# B&R Automation Studio project NAINV104C00R8L515F00 (part 12)

#### Act_OptP0923FullMask.st
```iecst
ACTION Act_OptP0923FullMask:

	IF eCurrPage = UIP0923Stopper THEN

		IF p_tyDI.bEStopSig = FALSE THEN
			p_tyC0002FullMask ACCESS ADR(tyP0923Stopper.tyFullMaskEStop);

		ELSIF p_tyDI.bCoverSWSig = FALSE THEN
			p_tyC0002FullMask ACCESS ADR(tyP0923Stopper.tyFullMaskCWSig);

		ELSIF p_tyDI.bSafetyRlySig = FALSE THEN
			p_tyC0002FullMask ACCESS ADR(tyP0923Stopper.tyFullMaskSafetyRly);

		ELSE
			p_tyC0002FullMask ACCESS ADR(tyP0923Stopper.tyFullMaskHide);

		END_IF

	END_IF

END_ACTION
```

#### Act_OptP0923Navi.st
```iecst
ACTION Act_OptP0923Navi:

	IF tyP0923Stopper.tyNaviBack.tyBtnBack.bRtCompl = TRUE THEN
		tyP0923Stopper.tyNaviBack.tyBtnBack.bRtCompl 	:= FALSE;
		tyP0923Stopper.tyNaviBack.tyBtnBack.bValue		:= FALSE;

		eChgPage	:= UIP0920MtrNPneuCtrl;

	END_IF

END_ACTION
```

#### Act_OptP0923ChgLyr.st
```iecst
ACTION Act_OptP0923ChgLyr:

	IF tyP0923Stopper.tyCom.tyBtnDCCtrl.bRtCompl = TRUE THEN
		tyP0923Stopper.tyCom.tyBtnDCCtrl.bRtCompl := FALSE;

		IF tyP0923Stopper.tyCom.tyBtnDCCtrl.bValue = TRUE THEN
			fUIInRtStatOff(ADR(tyP0923Stopper.tyDC.tyLyr.uiRtStat));
			fUIInRtStatHide(ADR(tyP0923Stopper.tyFB.tyLyr.uiRtStat));
		ELSE
			fUIInRtStatHide(ADR(tyP0923Stopper.tyDC.tyLyr.uiRtStat));
			fUIInRtStatOff(ADR(tyP0923Stopper.tyFB.tyLyr.uiRtStat));
		END_IF
	END_IF

END_ACTION
```

#### Act_OptP0923UpdtData.st
```iecst
ACTION Act_OptP0923UpdtData:

	//Update Bitmap
	IF p_bStopperExtCtrl THEN
		tyP0923Stopper.tyCom.tyBitmapMc.usiValueIdx	:= 1;
	ELSE
		tyP0923Stopper.tyCom.tyBitmapMc.usiValueIdx	:= 0;
	END_IF

END_ACTION
```

#### Act_OptP0923FBCtrl.st
```iecst
ACTION Act_OptP0923FBCtrl:

	IF tyP0923Stopper.tyCom.tyBtnDCCtrl.bValue = FALSE THEN

		//Control
		IF tyP0923Stopper.tyFB.tyBtnRetract.bRtCompl = TRUE THEN
			tyP0923Stopper.tyFB.tyBtnRetract.bRtCompl	:= FALSE;

			tyP0923Stopper.tyFB.tyBtnRetract.bValue		:= TRUE;
			tyP0923Stopper.tyFB.tyBtnExtend.bValue		:= FALSE;

		ELSIF tyP0923Stopper.tyFB.tyBtnExtend.bRtCompl = TRUE THEN
			tyP0923Stopper.tyFB.tyBtnExtend.bRtCompl	:= FALSE;

			tyP0923Stopper.tyFB.tyBtnExtend.bValue		:= TRUE;
			tyP0923Stopper.tyFB.tyBtnRetract.bValue		:= FALSE;

		END_IF

		//Action
		IF tyP0923Stopper.tyFB.tyBtnRetract.bValue = TRUE THEN
			eStopperAct	:= PneuActRet;

			IF p_eStopperStat = PneuActRet AND p_eStopperStatus = Done THEN
				eStopperAct	:= PneuActIdle;

				tyP0923Stopper.tyCom.tyBitmapMc.usiValueIdx	:= 0;
				tyP0923Stopper.tyFB.tyBtnRetract.bValue	:= FALSE;

			ELSIF p_eStopperStatus = Error THEN
				tyP0923Stopper.tyFB.tyBtnRetract.bValue	:= FALSE;

			END_IF

		ELSIF tyP0923Stopper.tyFB.tyBtnExtend.bValue = TRUE THEN
			eStopperAct	:= PneuActExt;

			IF p_eStopperStat = PneuActExt AND p_eStopperStatus = Done THEN
				eStopperAct	:= PneuActIdle;

				tyP0923Stopper.tyCom.tyBitmapMc.usiValueIdx	:= 1;
				tyP0923Stopper.tyFB.tyBtnExtend.bValue := FALSE;

			ELSIF p_eStopperStatus = Error THEN
				tyP0923Stopper.tyFB.tyBtnExtend.bValue := FALSE;

			END_IF
		END_IF

		//Update Status
		tyP0923Stopper.tyDC.tyBtnRetract.bRtCompl	:= FALSE;
		tyP0923Stopper.tyDC.tyBtnExtend.bRtCompl	:= FALSE;
		tyP0923Stopper.tyDC.tyBtnRetract.bValue		:= p_bStopperRetCtrl;
		tyP0923Stopper.tyDC.tyBtnExtend.bValue		:= p_bStopperExtCtrl;

		IF p_tyUsrMgmtCurrAccessRgt.bManualFBOnly THEN
			fUIInRtStatOff(ADR(tyP0923Stopper.tyCom.tyBtnDCCtrl.uiMaskRtStat));
		ELSE
			fUIInRtStatHide(ADR(tyP0923Stopper.tyCom.tyBtnDCCtrl.uiMaskRtStat));
		END_IF

	END_IF

END_ACTION
```

#### Act_OptP0923FBStat.st
```iecst
ACTION Act_OptP0923FBStat:

	tyP0923Stopper.tyFB.tyStringStat.sValue	:= p_sStopperStatTxt;

END_ACTION
```

#### Act_OptP0923DCCtrl.st
```iecst
ACTION Act_OptP0923DCCtrl:

	IF tyP0923Stopper.tyCom.tyBtnDCCtrl.bValue = TRUE THEN

		IF p_bStopperTwoCtrlOut = FALSE THEN

			IF tyP0923Stopper.tyDC.tyBtnRetract.bRtCompl = TRUE THEN
				tyP0923Stopper.tyDC.tyBtnRetract.bValue	:= TRUE;
				tyP0923Stopper.tyDC.tyBtnExtend.bValue	:= FALSE;

				eStopperAct	:= PneuActSetRet;

				IF p_eStopperStat = PneuActSetRet AND p_eStopperStatus = Done THEN
					eStopperAct	:= PneuActIdle;

					tyP0923Stopper.tyCom.tyBitmapMc.usiValueIdx	:= 0;
					tyP0923Stopper.tyDC.tyBtnRetract.bRtCompl	:= FALSE;
				END_IF

			ELSIF tyP0923Stopper.tyDC.tyBtnExtend.bRtCompl = TRUE THEN
				tyP0923Stopper.tyDC.tyBtnExtend.bValue	:= TRUE;
				tyP0923Stopper.tyDC.tyBtnRetract.bValue	:= FALSE;

				eStopperAct	:= PneuActSetExt;

				IF p_eStopperStat = PneuActSetExt AND p_eStopperStatus = Done THEN
					eStopperAct	:= PneuActIdle;

					tyP0923Stopper.tyCom.tyBitmapMc.usiValueIdx	:= 1;
					tyP0923Stopper.tyDC.tyBtnExtend.bRtCompl	:= FALSE;
				END_IF
			END_IF

		ELSE

			IF (tyP0923Stopper.tyDC.tyBtnRetract.bRtCompl = TRUE) OR (tyP0923Stopper.tyDC.tyBtnExtend.bRtCompl = TRUE) THEN
				IF (tyP0923Stopper.tyDC.tyBtnRetract.bValue = TRUE) AND (tyP0923Stopper.tyDC.tyBtnExtend.bValue = TRUE) THEN
					eStopperAct	:= PneuActSetAll;

					IF p_eStopperStat = PneuActSetAll AND p_eStopperStatus = Done THEN
						eStopperAct	:= PneuActIdle;

						tyP0923Stopper.tyDC.tyBtnRetract.bRtCompl	:= FALSE;
						tyP0923Stopper.tyDC.tyBtnExtend.bRtCompl	:= FALSE;
					END_IF

				ELSIF (tyP0923Stopper.tyDC.tyBtnRetract.bValue = TRUE) AND (tyP0923Stopper.tyDC.tyBtnExtend.bValue = FALSE) THEN
					eStopperAct	:= PneuActSetRet;

					IF p_eStopperStat = PneuActSetRet AND p_eStopperStatus = Done THEN
						eStopperAct	:= PneuActIdle;

						tyP0923Stopper.tyCom.tyBitmapMc.usiValueIdx	:= 0;
						tyP0923Stopper.tyDC.tyBtnRetract.bRtCompl	:= FALSE;
						tyP0923Stopper.tyDC.tyBtnExtend.bRtCompl	:= FALSE;
					END_IF

				ELSIF (tyP0923Stopper.tyDC.tyBtnRetract.bValue = FALSE) AND (tyP0923Stopper.tyDC.tyBtnExtend.bValue = TRUE) THEN
					eStopperAct	:= PneuActSetExt;

					IF p_eStopperStat = PneuActSetExt AND p_eStopperStatus = Done THEN
						eStopperAct	:= PneuActIdle;

						tyP0923Stopper.tyCom.tyBitmapMc.usiValueIdx	:= 1;
						tyP0923Stopper.tyDC.tyBtnRetract.bRtCompl	:= FALSE;
						tyP0923Stopper.tyDC.tyBtnExtend.bRtCompl	:= FALSE;
					END_IF

				ELSE
					eStopperAct	:= PneuActRstAll;

					IF p_eStopperStat = PneuActRstAll AND p_eStopperStatus = Done THEN
						eStopperAct	:= PneuActIdle;

						tyP0923Stopper.tyDC.tyBtnRetract.bRtCompl	:= FALSE;
						tyP0923Stopper.tyDC.tyBtnExtend.bRtCompl	:= FALSE;
					END_IF

				END_IF

			END_IF

		END_IF

		tyP0923Stopper.tyFB.tyBtnExtend.bRtCompl	:= FALSE;
		tyP0923Stopper.tyFB.tyBtnExtend.bValue		:= FALSE;
		tyP0923Stopper.tyFB.tyBtnRetract.bRtCompl	:= FALSE;
		tyP0923Stopper.tyFB.tyBtnRetract.bValue		:= FALSE;

	END_IF

END_ACTION
```

#### Act_OptP0923RstMnl.st
```iecst
ACTION Act_OptP0923RstMnl:

	IF EDGEPOS(p_eStopperStatus = Error) THEN

		eStopperAct	:= PneuActIdle;

		tyP0923Stopper.tyDC.tyBtnRetract.bValue 	:= FALSE;
		tyP0923Stopper.tyDC.tyBtnRetract.bRtCompl 	:= FALSE;

		tyP0923Stopper.tyDC.tyBtnExtend.bValue 		:= FALSE;
		tyP0923Stopper.tyDC.tyBtnExtend.bRtCompl 	:= FALSE;

		tyP0923Stopper.tyFB.tyBtnRetract.bValue 	:= FALSE;
		tyP0923Stopper.tyFB.tyBtnRetract.bRtCompl 	:= FALSE;

		tyP0923Stopper.tyFB.tyBtnExtend.bValue 		:= FALSE;
		tyP0923Stopper.tyFB.tyBtnExtend.bRtCompl 	:= FALSE;

	END_IF

	//Reset to Function Block Layer
	IF EDGEPOS(bManualMod = FALSE) THEN
		tyP0923Stopper.tyCom.tyBtnDCCtrl.bValue := FALSE;

		fUIInRtStatHide(ADR(tyP0923Stopper.tyDC.tyLyr.uiRtStat));
		fUIInRtStatOff(ADR(tyP0923Stopper.tyFB.tyLyr.uiRtStat));

		eStopperAct	:= PneuActIdle;

		tyP0923Stopper.tyDC.tyBtnRetract.bValue 	:= FALSE;
		tyP0923Stopper.tyDC.tyBtnRetract.bRtCompl 	:= FALSE;

		tyP0923Stopper.tyDC.tyBtnExtend.bValue 		:= FALSE;
		tyP0923Stopper.tyDC.tyBtnExtend.bRtCompl 	:= FALSE;

		tyP0923Stopper.tyFB.tyBtnRetract.bValue 	:= FALSE;
		tyP0923Stopper.tyFB.tyBtnRetract.bRtCompl 	:= FALSE;

		tyP0923Stopper.tyFB.tyBtnExtend.bValue 		:= FALSE;
		tyP0923Stopper.tyFB.tyBtnExtend.bRtCompl 	:= FALSE;

	END_IF

END_ACTION
```

#### Act_EntP0924Disp.st
```iecst
ACTION Act_EntP0924Disp:

	//Access Address
	p_tyC0003DualMask ACCESS ADR(tyP0924ClampWithRS.tyDualMaskHide);

	p_tyC0004Navi ACCESS ADR(tyP0924ClampWithRS.tyNaviLyr1);

	p_tyC0005Main ACCESS ADR(tyCommon.tyMain);

	p_tyC0007Notif ACCESS ADR(tyCommon.tyNotif);

	p_tyC0008MsgBox ACCESS ADR(tyP0924ClampWithRS.tyMsgBoxHide);

	p_tyC0009Info ACCESS ADR(tyCommon.tyInfo);

	p_tyP0924Clamp1WithRSCom ACCESS ADR(tyP0924ClampWithRS.tyClamp1WithRSCom);
	p_tyP0924Clamp1WithRSDC ACCESS ADR(tyP0924ClampWithRS.tyClamp1WithRSDC);
	p_tyP0924Clamp1WithRSFB ACCESS ADR(tyP0924ClampWithRS.tyClamp1WithRSFB);
	p_tyP0924Clamp1WithRSDis ACCESS ADR(tyP0924ClampWithRS.tyClamp1WithRSDis);

	p_tyP0924Clamp2WithRSCom ACCESS ADR(tyP0924ClampWithRS.tyClamp2WithRSCom);
	p_tyP0924Clamp2WithRSDC ACCESS ADR(tyP0924ClampWithRS.tyClamp2WithRSDC);
	p_tyP0924Clamp2WithRSFB ACCESS ADR(tyP0924ClampWithRS.tyClamp2WithRSFB);
	p_tyP0924Clamp2WithRSDis ACCESS ADR(tyP0924ClampWithRS.tyClamp2WithRSDis);

	p_tyP0924Clamp3WithRSCom ACCESS ADR(tyP0924ClampWithRS.tyClamp3WithRSCom);
	p_tyP0924Clamp3WithRSDC ACCESS ADR(tyP0924ClampWithRS.tyClamp3WithRSDC);
	p_tyP0924Clamp3WithRSFB ACCESS ADR(tyP0924ClampWithRS.tyClamp3WithRSFB);
	p_tyP0924Clamp3WithRSDis ACCESS ADR(tyP0924ClampWithRS.tyClamp3WithRSDis);

	//Display
	tyP0924ClampWithRS.tyClamp1WithRSDis.tyLyr.uiRtStat.0	:= (p_tyNtParamCurr.bProjClampPrep);
	tyP0924ClampWithRS.tyClamp2WithRSDis.tyLyr.uiRtStat.0	:= (p_tyNtParamCurr.bProjClampPrep);
	tyP0924ClampWithRS.tyClamp3WithRSDis.tyLyr.uiRtStat.0	:= (p_tyNtParamCurr.bProjClampPrep);

	fUIInRtStatOff(ADR(tyP0924ClampWithRS.tyNaviLyr1.tyLyr.uiRtStat));
	fUIInRtStatHide(ADR(tyP0924ClampWithRS.tyNaviLyr2.tyLyr.uiRtStat));

	fUIInRtStatOff(ADR(tyP0924ClampWithRS.tyClamp1WithRSCom.tyLyr.uiRtStat));
	fUIInRtStatOff(ADR(tyP0924ClampWithRS.tyClamp2WithRSCom.tyLyr.uiRtStat));

	fUIInRtStatHide(ADR(tyP0924ClampWithRS.tyClamp3WithRSCom.tyLyr.uiRtStat));
	fUIInRtStatHide(ADR(tyP0924ClampWithRS.tyClamp3WithRSDC.tyLyr.uiRtStat));
	fUIInRtStatHide(ADR(tyP0924ClampWithRS.tyClamp3WithRSFB.tyLyr.uiRtStat));
	fUIInRtStatHide(ADR(tyP0924ClampWithRS.tyClamp3WithRSDis.tyLyr.uiRtStat));

	//Display
	IF tyP0924ClampWithRS.tyClamp1WithRSCom.tyBtnSwitch.bValue = TRUE THEN
		fUIInRtStatOff(ADR(tyP0924ClampWithRS.tyClamp1WithRSDC.tyLyr.uiRtStat));
		fUIInRtStatHide(ADR(tyP0924ClampWithRS.tyClamp1WithRSFB.tyLyr.uiRtStat));
	ELSE
		fUIInRtStatOff(ADR(tyP0924ClampWithRS.tyClamp1WithRSFB.tyLyr.uiRtStat));
		fUIInRtStatHide(ADR(tyP0924ClampWithRS.tyClamp1WithRSDC.tyLyr.uiRtStat));
	END_IF

	IF tyP0924ClampWithRS.tyClamp2WithRSCom.tyBtnSwitch.bValue = TRUE THEN
		fUIInRtStatOff(ADR(tyP0924ClampWithRS.tyClamp2WithRSDC.tyLyr.uiRtStat));
		fUIInRtStatHide(ADR(tyP0924ClampWithRS.tyClamp2WithRSFB.tyLyr.uiRtStat));
	ELSE
		fUIInRtStatOff(ADR(tyP0924ClampWithRS.tyClamp2WithRSFB.tyLyr.uiRtStat));
		fUIInRtStatHide(ADR(tyP0924ClampWithRS.tyClamp2WithRSDC.tyLyr.uiRtStat));
	END_IF

//	IF tyP0924ClampWithRS.tyClamp3WithRSCom.tyBtnSwitch.bValue = TRUE THEN
//		fUIInRtStatOff(ADR(tyP0924ClampWithRS.tyClamp3WithRSDC.tyLyr.uiRtStat));
//		fUIInRtStatHide(ADR(tyP0924ClampWithRS.tyClamp3WithRSFB.tyLyr.uiRtStat));
//	ELSE
//		fUIInRtStatOff(ADR(tyP0924ClampWithRS.tyClamp3WithRSFB.tyLyr.uiRtStat));
//		fUIInRtStatHide(ADR(tyP0924ClampWithRS.tyClamp3WithRSDC.tyLyr.uiRtStat));
//	END_IF

END_ACTION
```

#### Act_OptP0924Navi.st
```iecst
ACTION Act_OptP0924Navi:

	IF tyP0924ClampWithRS.tyNaviLyr1.tyBtnBack.bRtCompl = TRUE OR tyP0924ClampWithRS.tyNaviLyr2.tyBtnBack.bRtCompl = TRUE THEN
		tyP0924ClampWithRS.tyNaviLyr1.tyBtnBack.bRtCompl	:= FALSE;
		tyP0924ClampWithRS.tyNaviLyr2.tyBtnBack.bRtCompl	:= FALSE;

		eChgPage	:= UIP0920MtrNPneuCtrl;

	ELSIF tyP0924ClampWithRS.tyNaviLyr1.tyBtnLeft.bRtCompl = TRUE OR tyP0924ClampWithRS.tyNaviLyr1.tyBtnRgt.bRtCompl = TRUE THEN
		tyP0924ClampWithRS.tyNaviLyr1.tyBtnLeft.bRtCompl	:= FALSE;
		tyP0924ClampWithRS.tyNaviLyr1.tyBtnRgt.bRtCompl	:= FALSE;

		p_tyC0004Navi ACCESS ADR(tyP0924ClampWithRS.tyNaviLyr2);

		fUIInRtStatHide(ADR(tyP0924ClampWithRS.tyNaviLyr1.tyLyr.uiRtStat));
		fUIInRtStatOff(ADR (tyP0924ClampWithRS.tyNaviLyr2.tyLyr.uiRtStat));
		fUIInRtStatOff(ADR(tyP0924ClampWithRS.tyClamp3WithRSCom.tyLyr.uiRtStat));

		fUIInRtStatHide(ADR (tyP0924ClampWithRS.tyClamp1WithRSCom.tyLyr.uiRtStat));
		fUIInRtStatHide(ADR (tyP0924ClampWithRS.tyClamp1WithRSDC.tyLyr.uiRtStat));
		fUIInRtStatHide(ADR (tyP0924ClampWithRS.tyClamp1WithRSFB.tyLyr.uiRtStat));
		fUIInRtStatHide(ADR (tyP0924ClampWithRS.tyClamp2WithRSCom.tyLyr.uiRtStat));
		fUIInRtStatHide(ADR (tyP0924ClampWithRS.tyClamp2WithRSDC.tyLyr.uiRtStat));
		fUIInRtStatHide(ADR (tyP0924ClampWithRS.tyClamp2WithRSFB.tyLyr.uiRtStat));

		IF tyP0924ClampWithRS.tyClamp3WithRSCom.tyBtnSwitch.bValue = TRUE THEN
			fUIInRtStatOff(ADR(tyP0924ClampWithRS.tyClamp3WithRSDC.tyLyr.uiRtStat));
			fUIInRtStatHide(ADR(tyP0924ClampWithRS.tyClamp3WithRSFB.tyLyr.uiRtStat));
		ELSE
			fUIInRtStatOff(ADR(tyP0924ClampWithRS.tyClamp3WithRSFB.tyLyr.uiRtStat));
			fUIInRtStatHide(ADR(tyP0924ClampWithRS.tyClamp3WithRSDC.tyLyr.uiRtStat));
		END_IF

	ELSIF tyP0924ClampWithRS.tyNaviLyr2.tyBtnLeft.bRtCompl = TRUE OR tyP0924ClampWithRS.tyNaviLyr2.tyBtnRgt.bRtCompl = TRUE THEN
		tyP0924ClampWithRS.tyNaviLyr2.tyBtnLeft.bRtCompl	:= FALSE;
		tyP0924ClampWithRS.tyNaviLyr2.tyBtnRgt.bRtCompl	:= FALSE;

		p_tyC0004Navi ACCESS ADR(tyP0924ClampWithRS.tyNaviLyr1);

		fUIInRtStatOff(ADR(tyP0924ClampWithRS.tyNaviLyr1.tyLyr.uiRtStat));
		fUIInRtStatHide(ADR(tyP0924ClampWithRS.tyNaviLyr2.tyLyr.uiRtStat));
		fUIInRtStatHide(ADR(tyP0924ClampWithRS.tyClamp3WithRSFB.tyLyr.uiRtStat));
		fUIInRtStatHide(ADR(tyP0924ClampWithRS.tyClamp3WithRSDC.tyLyr.uiRtStat));
		fUIInRtStatHide(ADR(tyP0924ClampWithRS.tyClamp3WithRSCom.tyLyr.uiRtStat));

		fUIInRtStatOff(ADR(tyP0924ClampWithRS.tyClamp1WithRSCom.tyLyr.uiRtStat));
		fUIInRtStatOff(ADR(tyP0924ClampWithRS.tyClamp2WithRSCom.tyLyr.uiRtStat));

		IF tyP0924ClampWithRS.tyClamp1WithRSCom.tyBtnSwitch.bValue = TRUE THEN
			fUIInRtStatOff(ADR(tyP0924ClampWithRS.tyClamp1WithRSDC.tyLyr.uiRtStat));
			fUIInRtStatHide(ADR(tyP0924ClampWithRS.tyClamp1WithRSFB.tyLyr.uiRtStat));
		ELSE
			fUIInRtStatOff(ADR(tyP0924ClampWithRS.tyClamp1WithRSFB.tyLyr.uiRtStat));
			fUIInRtStatHide(ADR(tyP0924ClampWithRS.tyClamp1WithRSDC.tyLyr.uiRtStat));
		END_IF

		IF tyP0924ClampWithRS.tyClamp2WithRSCom.tyBtnSwitch.bValue = TRUE THEN
			fUIInRtStatOff(ADR(tyP0924ClampWithRS.tyClamp2WithRSDC.tyLyr.uiRtStat));
			fUIInRtStatHide(ADR(tyP0924ClampWithRS.tyClamp2WithRSFB.tyLyr.uiRtStat));
		ELSE
			fUIInRtStatOff(ADR(tyP0924ClampWithRS.tyClamp2WithRSFB.tyLyr.uiRtStat));
			fUIInRtStatHide(ADR(tyP0924ClampWithRS.tyClamp2WithRSDC.tyLyr.uiRtStat));
		END_IF

	END_IF

END_ACTION
```

#### Act_OptP0924DualMask.st
```iecst
ACTION Act_OptP0924DualMask:

	IF eCurrPage = UIP0924ClampWithRS THEN

		IF p_tyDI.bEStopSig = FALSE THEN
			p_tyC0003DualMask ACCESS ADR(tyP0924ClampWithRS.tyDualMaskEStop);

			IF 	tyP0924ClampWithRS.tyNaviLyr1.tyLyr.uiRtStat.0=FALSE THEN
				tyP0924ClampWithRS.tyDualMaskEStop.tyBtnLeftMask.uiMaskRtStat.0	:= FALSE ;
				tyP0924ClampWithRS.tyDualMaskEStop.tyBtnRgtMask.uiMaskRtStat.0	:= FALSE;
			ELSE
				tyP0924ClampWithRS.tyDualMaskEStop.tyBtnLeftMask.uiMaskRtStat.0	:= FALSE ;
				tyP0924ClampWithRS.tyDualMaskEStop.tyBtnRgtMask.uiMaskRtStat.0	:= TRUE;
			END_IF

		ELSIF p_tyDI.bCoverSWSig = FALSE THEN
			p_tyC0003DualMask ACCESS ADR(tyP0924ClampWithRS.tyDualMaskCWSig);

			IF 	tyP0924ClampWithRS.tyNaviLyr1.tyLyr.uiRtStat.0=FALSE THEN
				tyP0924ClampWithRS.tyDualMaskEStop.tyBtnLeftMask.uiMaskRtStat.0	:= FALSE ;
				tyP0924ClampWithRS.tyDualMaskEStop.tyBtnRgtMask.uiMaskRtStat.0	:= FALSE;
			ELSE
				tyP0924ClampWithRS.tyDualMaskEStop.tyBtnLeftMask.uiMaskRtStat.0	:= FALSE ;
				tyP0924ClampWithRS.tyDualMaskEStop.tyBtnRgtMask.uiMaskRtStat.0	:= TRUE;
			END_IF

		ELSIF p_tyDI.bSafetyRlySig = FALSE THEN
			p_tyC0003DualMask ACCESS ADR(tyP0924ClampWithRS.tyDualMaskSafetyRly);

			IF 	tyP0924ClampWithRS.tyNaviLyr1.tyLyr.uiRtStat.0=FALSE THEN
				tyP0924ClampWithRS.tyDualMaskEStop.tyBtnLeftMask.uiMaskRtStat.0	:= FALSE ;
				tyP0924ClampWithRS.tyDualMaskEStop.tyBtnRgtMask.uiMaskRtStat.0	:= FALSE;
			ELSE
				tyP0924ClampWithRS.tyDualMaskEStop.tyBtnLeftMask.uiMaskRtStat.0	:= FALSE ;
				tyP0924ClampWithRS.tyDualMaskEStop.tyBtnRgtMask.uiMaskRtStat.0	:= TRUE;
			END_IF

		ELSIF p_eAWOpenStatus = Busy THEN
			p_tyC0003DualMask ACCESS ADR(tyP0924ClampWithRS.tyDualMaskAWMovInterrupt);

			IF 	tyP0924ClampWithRS.tyNaviLyr1.tyLyr.uiRtStat.0=FALSE THEN
				tyP0924ClampWithRS.tyDualMaskEStop.tyBtnLeftMask.uiMaskRtStat.0	:= FALSE ;
				tyP0924ClampWithRS.tyDualMaskEStop.tyBtnRgtMask.uiMaskRtStat.0	:= FALSE;
			ELSE
				tyP0924ClampWithRS.tyDualMaskEStop.tyBtnLeftMask.uiMaskRtStat.0	:= FALSE ;
				tyP0924ClampWithRS.tyDualMaskEStop.tyBtnRgtMask.uiMaskRtStat.0	:= TRUE;
			END_IF

		ELSE
			p_tyC0003DualMask ACCESS ADR(tyP0924ClampWithRS.tyDualMaskHide);

		END_IF

	END_IF

END_ACTION
```

#### Act_OptP0924Clamp1ChgLyr.st
```iecst
ACTION Act_OptP0924Clamp1ChgLyr:

	IF tyP0924ClampWithRS.tyClamp1WithRSCom.tyBtnSwitch.bRtCompl THEN
		tyP0924ClampWithRS.tyClamp1WithRSCom.tyBtnSwitch.bRtCompl := FALSE;

		IF tyP0924ClampWithRS.tyClamp1WithRSCom.tyBtnSwitch.bValue = TRUE THEN
			fUIInRtStatOff(ADR(tyP0924ClampWithRS.tyClamp1WithRSDC.tyLyr.uiRtStat));
			fUIInRtStatHide(ADR(tyP0924ClampWithRS.tyClamp1WithRSFB.tyLyr.uiRtStat));
		ELSE
			fUIInRtStatHide(ADR(tyP0924ClampWithRS.tyClamp1WithRSDC.tyLyr.uiRtStat));
			fUIInRtStatOff(ADR(tyP0924ClampWithRS.tyClamp1WithRSFB.tyLyr.uiRtStat));
		END_IF

	END_IF

END_ACTION
```

#### Act_OptP0924Clamp1Sen.st
```iecst
ACTION Act_OptP0924Clamp1Sen:

	tyP0924ClampWithRS.tyClamp1WithRSCom.tyBtnClampRS.bValue		:= p_tyDI.bClampRS1;
	tyP0924ClampWithRS.tyClamp1WithRSCom.tyBtnUnClampRS.bValue		:= p_tyDI.bUnClampRS1;

	//Machine Bitmap
	IF p_tyDI.bClampRS1 = TRUE THEN
		tyP0924ClampWithRS.tyClamp1WithRSCom.tyBitmapMc.usiValueIdx	:= 1;
	ELSE
		tyP0924ClampWithRS.tyClamp1WithRSCom.tyBitmapMc.usiValueIdx	:= 0;
	END_IF

END_ACTION
```

#### Act_OptP0924Clamp1FB.st
```iecst
ACTION Act_OptP0924Clamp1FB:

	IF tyP0924ClampWithRS.tyClamp1WithRSCom.tyBtnSwitch.bValue = FALSE THEN

		IF tyP0924ClampWithRS.tyClamp1WithRSFB.tyBtnExt.bRtCompl = TRUE THEN
			tyP0924ClampWithRS.tyClamp1WithRSFB.tyBtnExt.bRtCompl	:= FALSE;

			tyP0924ClampWithRS.tyClamp1WithRSFB.tyBtnExt.bValue	:= TRUE;
			tyP0924ClampWithRS.tyClamp1WithRSFB.tyBtnRet.bValue	:= FALSE;

		ELSIF tyP0924ClampWithRS.tyClamp1WithRSFB.tyBtnRet.bRtCompl = TRUE THEN
			tyP0924ClampWithRS.tyClamp1WithRSFB.tyBtnRet.bRtCompl	:= FALSE;

			tyP0924ClampWithRS.tyClamp1WithRSFB.tyBtnRet.bValue	:= TRUE;
			tyP0924ClampWithRS.tyClamp1WithRSFB.tyBtnExt.bValue	:= FALSE;
		END_IF

		IF tyP0924ClampWithRS.tyClamp1WithRSFB.tyBtnExt.bValue = TRUE THEN
			eClamp1Act	:= PneuActExt;

			IF p_eClamp1Stat = PneuActExt AND p_eClamp1Status = Done THEN
				eClamp1Act	:= PneuActIdle;

				tyP0924ClampWithRS.tyClamp1WithRSFB.tyBtnExt.bValue	:= FALSE;

			ELSIF p_eClamp1Status = Error THEN
				tyP0924ClampWithRS.tyClamp1WithRSFB.tyBtnExt.bValue	:= FALSE;
			END_IF

		ELSIF tyP0924ClampWithRS.tyClamp1WithRSFB.tyBtnRet.bValue = TRUE THEN
			eClamp1Act	:= PneuActRet;

			IF p_eClamp1Stat = PneuActRet AND p_eClamp1Status = Done THEN
				eClamp1Act	:= PneuActIdle;

				tyP0924ClampWithRS.tyClamp1WithRSFB.tyBtnRet.bValue := FALSE;
			ELSIF p_eClamp1Status = Error THEN
				tyP0924ClampWithRS.tyClamp1WithRSFB.tyBtnRet.bValue := FALSE;
			END_IF
		END_IF

		//Update Direct Control Status
		tyP0924ClampWithRS.tyClamp1WithRSDC.tyBtnExt.bRtCompl	:= FALSE;
		tyP0924ClampWithRS.tyClamp1WithRSDC.tyBtnRet.bRtCompl	:= FALSE;
		tyP0924ClampWithRS.tyClamp1WithRSDC.tyBtnExt.bValue		:= p_bClamp1ExtCtrl;
		tyP0924ClampWithRS.tyClamp1WithRSDC.tyBtnRet.bValue		:= p_bClamp1RetCtrl;

		IF p_tyUsrMgmtCurrAccessRgt.bManualFBOnly THEN
			fUIInRtStatOff(ADR(tyP0924ClampWithRS.tyClamp1WithRSCom.tyBtnSwitch.uiMaskRtStat));
		ELSE
			fUIInRtStatHide(ADR(tyP0924ClampWithRS.tyClamp1WithRSCom.tyBtnSwitch.uiMaskRtStat));
		END_IF

	END_IF

END_ACTION
```

#### Act_OptP0924Clamp1FBStat.st
```iecst
ACTION Act_OptP0924Clamp1FBStat:

	tyP0924ClampWithRS.tyClamp1WithRSFB.tyStringStat.sValue	:= p_sClamp1StatTxt;

END_ACTION
```

#### Act_OptP0924Clamp1DC.st
```iecst
ACTION Act_OptP0924Clamp1DC:

	IF tyP0924ClampWithRS.tyClamp1WithRSCom.tyBtnSwitch.bValue = TRUE THEN
		IF p_bClamp1TwoCtrlOut = FALSE THEN
			IF tyP0924ClampWithRS.tyClamp1WithRSDC.tyBtnExt.bRtCompl = TRUE THEN
				tyP0924ClampWithRS.tyClamp1WithRSDC.tyBtnExt.bValue	:= TRUE;
				tyP0924ClampWithRS.tyClamp1WithRSDC.tyBtnRet.bValue	:= FALSE;

				eClamp1Act	:= PneuActSetExt;

				IF p_eClamp1Stat = PneuActSetExt AND p_eClamp1Status = Done THEN
					eClamp1Act	:= PneuActIdle;

					tyP0924ClampWithRS.tyClamp1WithRSDC.tyBtnExt.bRtCompl	:= FALSE;
				END_IF

			ELSIF tyP0924ClampWithRS.tyClamp1WithRSDC.tyBtnRet.bRtCompl = TRUE THEN
				tyP0924ClampWithRS.tyClamp1WithRSDC.tyBtnRet.bValue	:= TRUE;
				tyP0924ClampWithRS.tyClamp1WithRSDC.tyBtnExt.bValue	:= FALSE;

				eClamp1Act	:= PneuActSetRet;

				IF p_eClamp1Stat = PneuActSetRet AND p_eClamp1Status = Done THEN
					eClamp1Act	:= PneuActIdle;

					tyP0924ClampWithRS.tyClamp1WithRSDC.tyBtnRet.bRtCompl	:= FALSE;
				END_IF
			END_IF

		ELSE
			IF (tyP0924ClampWithRS.tyClamp1WithRSDC.tyBtnExt.bRtCompl = TRUE) OR (tyP0924ClampWithRS.tyClamp1WithRSDC.tyBtnRet.bRtCompl = TRUE) THEN
				IF (tyP0924ClampWithRS.tyClamp1WithRSDC.tyBtnExt.bValue = TRUE) AND (tyP0924ClampWithRS.tyClamp1WithRSDC.tyBtnRet.bValue = TRUE) THEN
					eClamp1Act	:= PneuActSetAll;

					IF p_eClamp1Stat = PneuActSetAll AND p_eClamp1Status = Done THEN
						eClamp1Act	:= PneuActIdle;

						tyP0924ClampWithRS.tyClamp1WithRSDC.tyBtnExt.bRtCompl	:= FALSE;
						tyP0924ClampWithRS.tyClamp1WithRSDC.tyBtnRet.bRtCompl	:= FALSE;
					END_IF

				ELSIF (tyP0924ClampWithRS.tyClamp1WithRSDC.tyBtnExt.bValue = TRUE) AND (tyP0924ClampWithRS.tyClamp1WithRSDC.tyBtnRet.bValue = FALSE) THEN
					eClamp1Act	:= PneuActSetExt;

					IF p_eClamp1Stat = PneuActSetExt AND p_eClamp1Status = Done THEN
						eClamp1Act	:= PneuActIdle;

						tyP0924ClampWithRS.tyClamp1WithRSDC.tyBtnExt.bRtCompl	:= FALSE;
						tyP0924ClampWithRS.tyClamp1WithRSDC.tyBtnRet.bRtCompl	:= FALSE;
					END_IF

				ELSIF (tyP0924ClampWithRS.tyClamp1WithRSDC.tyBtnExt.bValue = FALSE) AND (tyP0924ClampWithRS.tyClamp1WithRSDC.tyBtnRet.bValue = TRUE) THEN
					eClamp1Act	:= PneuActSetRet;

					IF p_eClamp1Stat = PneuActSetRet AND p_eClamp1Status = Done THEN
						eClamp1Act	:= PneuActIdle;

						tyP0924ClampWithRS.tyClamp1WithRSDC.tyBtnExt.bRtCompl	:= FALSE;
						tyP0924ClampWithRS.tyClamp1WithRSDC.tyBtnRet.bRtCompl	:= FALSE;
					END_IF

				ELSE
					eClamp1Act	:= PneuActRstAll;

					IF p_eClamp1Stat = PneuActRstAll AND p_eClamp1Status = Done THEN
						eClamp1Act	:= PneuActIdle;

						tyP0924ClampWithRS.tyClamp1WithRSDC.tyBtnExt.bRtCompl	:= FALSE;
						tyP0924ClampWithRS.tyClamp1WithRSDC.tyBtnRet.bRtCompl	:= FALSE;
					END_IF

				END_IF
			END_IF
		END_IF

		tyP0924ClampWithRS.tyClamp1WithRSFB.tyBtnRet.bRtCompl	:= FALSE;
		tyP0924ClampWithRS.tyClamp1WithRSFB.tyBtnRet.bValue	:= FALSE;
		tyP0924ClampWithRS.tyClamp1WithRSFB.tyBtnExt.bRtCompl	:= FALSE;
		tyP0924ClampWithRS.tyClamp1WithRSFB.tyBtnExt.bValue	:= FALSE;

	END_IF

END_ACTION
```

#### Act_OptP0924Clamp2ChgLyr.st
```iecst
ACTION Act_OptP0924Clamp2ChgLyr:

	IF	tyP0924ClampWithRS.tyClamp2WithRSCom.tyBtnSwitch.bRtCompl THEN
		tyP0924ClampWithRS.tyClamp2WithRSCom.tyBtnSwitch.bRtCompl := FALSE;

		IF tyP0924ClampWithRS.tyClamp2WithRSCom.tyBtnSwitch.bValue = TRUE THEN
			fUIInRtStatOff(ADR(tyP0924ClampWithRS.tyClamp2WithRSDC.tyLyr.uiRtStat));
			fUIInRtStatHide(ADR(tyP0924ClampWithRS.tyClamp2WithRSFB.tyLyr.uiRtStat));
		ELSE
			fUIInRtStatHide(ADR(tyP0924ClampWithRS.tyClamp2WithRSDC.tyLyr.uiRtStat));
			fUIInRtStatOff(ADR(tyP0924ClampWithRS.tyClamp2WithRSFB.tyLyr.uiRtStat));
		END_IF

	END_IF

END_ACTION
```

#### Act_OptP0924Clamp2Sen.st
```iecst
ACTION Act_OptP0924Clamp2Sen:

	tyP0924ClampWithRS.tyClamp2WithRSCom.tyBtnClampRS.bValue		:= p_tyDI.bClampRS2;
	tyP0924ClampWithRS.tyClamp2WithRSCom.tyBtnUnClampRS.bValue		:= p_tyDI.bUnClampRS2;

	//Machine Bitmap
	IF p_tyDI.bClampRS2 = TRUE THEN
		tyP0924ClampWithRS.tyClamp2WithRSCom.tyBitmapMc.usiValueIdx	:= 1;
	ELSE
		tyP0924ClampWithRS.tyClamp2WithRSCom.tyBitmapMc.usiValueIdx	:= 0;
	END_IF

END_ACTION
```

#### Act_OptP0924Clamp2FB.st
```iecst
ACTION Act_OptP0924Clamp2FB:

	IF tyP0924ClampWithRS.tyClamp2WithRSCom.tyBtnSwitch.bValue = FALSE THEN

		IF tyP0924ClampWithRS.tyClamp2WithRSFB.tyBtnExt.bRtCompl = TRUE THEN
			tyP0924ClampWithRS.tyClamp2WithRSFB.tyBtnExt.bRtCompl	:= FALSE;

			tyP0924ClampWithRS.tyClamp2WithRSFB.tyBtnExt.bValue	:= TRUE;
			tyP0924ClampWithRS.tyClamp2WithRSFB.tyBtnRet.bValue	:= FALSE;

		ELSIF tyP0924ClampWithRS.tyClamp2WithRSFB.tyBtnRet.bRtCompl = TRUE THEN
			tyP0924ClampWithRS.tyClamp2WithRSFB.tyBtnRet.bRtCompl	:= FALSE;

			tyP0924ClampWithRS.tyClamp2WithRSFB.tyBtnRet.bValue	:= TRUE;
			tyP0924ClampWithRS.tyClamp2WithRSFB.tyBtnExt.bValue	:= FALSE;
		END_IF

		IF tyP0924ClampWithRS.tyClamp2WithRSFB.tyBtnExt.bValue = TRUE THEN
			eClamp2Act	:= PneuActExt;

			IF p_eClamp2Stat = PneuActExt AND p_eClamp2Status = Done THEN
				eClamp2Act	:= PneuActIdle;

				tyP0924ClampWithRS.tyClamp2WithRSFB.tyBtnExt.bValue	:= FALSE;

			ELSIF p_eClamp2Status = Error THEN
				tyP0924ClampWithRS.tyClamp2WithRSFB.tyBtnExt.bValue	:= FALSE;
			END_IF

		ELSIF tyP0924ClampWithRS.tyClamp2WithRSFB.tyBtnRet.bValue = TRUE THEN
			eClamp2Act	:= PneuActRet;

			IF p_eClamp2Stat = PneuActRet AND p_eClamp2Status = Done THEN
				eClamp2Act	:= PneuActIdle;

				tyP0924ClampWithRS.tyClamp2WithRSFB.tyBtnRet.bValue := FALSE;
			ELSIF p_eClamp2Status = Error THEN
				tyP0924ClampWithRS.tyClamp2WithRSFB.tyBtnRet.bValue := FALSE;
			END_IF
		END_IF

		//Update Direct Control Status
		tyP0924ClampWithRS.tyClamp2WithRSDC.tyBtnExt.bRtCompl	:= FALSE;
		tyP0924ClampWithRS.tyClamp2WithRSDC.tyBtnRet.bRtCompl	:= FALSE;
		tyP0924ClampWithRS.tyClamp2WithRSDC.tyBtnExt.bValue	:= p_bClamp2ExtCtrl;
		tyP0924ClampWithRS.tyClamp2WithRSDC.tyBtnRet.bValue	:= p_bClamp2RetCtrl;

		IF p_tyUsrMgmtCurrAccessRgt.bManualFBOnly THEN
			fUIInRtStatOff(ADR(tyP0924ClampWithRS.tyClamp2WithRSCom.tyBtnSwitch.uiMaskRtStat));
		ELSE
			fUIInRtStatHide(ADR(tyP0924ClampWithRS.tyClamp2WithRSCom.tyBtnSwitch.uiMaskRtStat));
		END_IF

	END_IF

END_ACTION
```

#### Act_OptP0924Clamp2FBStat.st
```iecst
ACTION Act_OptP0924Clamp2FBStat:

	tyP0924ClampWithRS.tyClamp2WithRSFB.tyStringStat.sValue	:= p_sClamp2StatTxt;

END_ACTION
```

#### Act_OptP0924Clamp2DC.st
```iecst
ACTION Act_OptP0924Clamp2DC:

	IF tyP0924ClampWithRS.tyClamp2WithRSCom.tyBtnSwitch.bValue = TRUE THEN
		IF p_bClamp1TwoCtrlOut = FALSE THEN
			IF tyP0924ClampWithRS.tyClamp2WithRSDC.tyBtnExt.bRtCompl = TRUE THEN
				tyP0924ClampWithRS.tyClamp2WithRSDC.tyBtnExt.bValue	:= TRUE;
				tyP0924ClampWithRS.tyClamp2WithRSDC.tyBtnRet.bValue	:= FALSE;

				eClamp2Act	:= PneuActSetExt;

				IF p_eClamp2Stat = PneuActSetExt AND p_eClamp2Status = Done THEN
					eClamp2Act	:= PneuActIdle;

					tyP0924ClampWithRS.tyClamp2WithRSDC.tyBtnExt.bRtCompl	:= FALSE;
				END_IF

			ELSIF tyP0924ClampWithRS.tyClamp2WithRSDC.tyBtnRet.bRtCompl = TRUE THEN
				tyP0924ClampWithRS.tyClamp2WithRSDC.tyBtnRet.bValue	:= TRUE;
				tyP0924ClampWithRS.tyClamp2WithRSDC.tyBtnExt.bValue	:= FALSE;

				eClamp2Act	:= PneuActSetRet;

				IF p_eClamp2Stat = PneuActSetRet AND p_eClamp2Status = Done THEN
					eClamp2Act	:= PneuActIdle;

					tyP0924ClampWithRS.tyClamp2WithRSDC.tyBtnRet.bRtCompl	:= FALSE;
				END_IF
			END_IF

		ELSE
			IF (tyP0924ClampWithRS.tyClamp2WithRSDC.tyBtnExt.bRtCompl = TRUE) OR (tyP0924ClampWithRS.tyClamp2WithRSDC.tyBtnRet.bRtCompl = TRUE) THEN
				IF (tyP0924ClampWithRS.tyClamp2WithRSDC.tyBtnExt.bValue = TRUE) AND (tyP0924ClampWithRS.tyClamp2WithRSDC.tyBtnRet.bValue = TRUE) THEN
					eClamp2Act	:= PneuActSetAll;

					IF p_eClamp2Stat = PneuActSetAll AND p_eClamp2Status = Done THEN
						eClamp2Act	:= PneuActIdle;

						tyP0924ClampWithRS.tyClamp2WithRSDC.tyBtnExt.bRtCompl	:= FALSE;
						tyP0924ClampWithRS.tyClamp2WithRSDC.tyBtnRet.bRtCompl	:= FALSE;
					END_IF

				ELSIF (tyP0924ClampWithRS.tyClamp2WithRSDC.tyBtnExt.bValue = TRUE) AND (tyP0924ClampWithRS.tyClamp2WithRSDC.tyBtnRet.bValue = FALSE) THEN
					eClamp2Act	:= PneuActSetExt;

					IF p_eClamp2Stat = PneuActSetExt AND p_eClamp2Status = Done THEN
						eClamp2Act	:= PneuActIdle;

						tyP0924ClampWithRS.tyClamp2WithRSDC.tyBtnExt.bRtCompl	:= FALSE;
						tyP0924ClampWithRS.tyClamp2WithRSDC.tyBtnRet.bRtCompl	:= FALSE;
					END_IF

				ELSIF (tyP0924ClampWithRS.tyClamp2WithRSDC.tyBtnExt.bValue = FALSE) AND (tyP0924ClampWithRS.tyClamp2WithRSDC.tyBtnRet.bValue = TRUE) THEN
					eClamp2Act	:= PneuActSetRet;

					IF p_eClamp2Stat = PneuActSetRet AND p_eClamp2Status = Done THEN
						eClamp2Act	:= PneuActIdle;

						tyP0924ClampWithRS.tyClamp2WithRSDC.tyBtnExt.bRtCompl	:= FALSE;
						tyP0924ClampWithRS.tyClamp2WithRSDC.tyBtnRet.bRtCompl	:= FALSE;
					END_IF

				ELSE
					eClamp2Act	:= PneuActRstAll;

					IF p_eClamp2Stat = PneuActRstAll AND p_eClamp2Status = Done THEN
						eClamp2Act	:= PneuActIdle;

						tyP0924ClampWithRS.tyClamp2WithRSDC.tyBtnExt.bRtCompl	:= FALSE;
						tyP0924ClampWithRS.tyClamp2WithRSDC.tyBtnRet.bRtCompl	:= FALSE;
					END_IF

				END_IF
			END_IF
		END_IF

		tyP0924ClampWithRS.tyClamp2WithRSFB.tyBtnRet.bRtCompl	:= FALSE;
		tyP0924ClampWithRS.tyClamp2WithRSFB.tyBtnRet.bValue		:= FALSE;
		tyP0924ClampWithRS.tyClamp2WithRSFB.tyBtnExt.bRtCompl	:= FALSE;
		tyP0924ClampWithRS.tyClamp2WithRSFB.tyBtnExt.bValue		:= FALSE;

	END_IF

END_ACTION
```

#### Act_OptP0924Clamp3ChgLyr.st
```iecst
ACTION Act_OptP0924Clamp3ChgLyr:

	IF tyP0924ClampWithRS.tyClamp3WithRSCom.tyBtnSwitch.bRtCompl THEN
		tyP0924ClampWithRS.tyClamp3WithRSCom.tyBtnSwitch.bRtCompl := FALSE;

		IF tyP0924ClampWithRS.tyClamp3WithRSCom.tyBtnSwitch.bValue = TRUE THEN
			fUIInRtStatOff(ADR(tyP0924ClampWithRS.tyClamp3WithRSDC.tyLyr.uiRtStat));
			fUIInRtStatHide(ADR(tyP0924ClampWithRS.tyClamp3WithRSFB.tyLyr.uiRtStat));
		ELSE
			fUIInRtStatHide(ADR(tyP0924ClampWithRS.tyClamp3WithRSDC.tyLyr.uiRtStat));
			fUIInRtStatOff(ADR(tyP0924ClampWithRS.tyClamp3WithRSFB.tyLyr.uiRtStat));
		END_IF

	END_IF

END_ACTION
```

#### Act_OptP0924Clamp3Sen.st
```iecst
ACTION Act_OptP0924Clamp3Sen:

	tyP0924ClampWithRS.tyClamp3WithRSCom.tyBtnClampRS.bValue		:= p_tyDI.bClampRS3;
	tyP0924ClampWithRS.tyClamp3WithRSCom.tyBtnUnClampRS.bValue	:= p_tyDI.bUnClampRS3;

	//Machine Bitmap
	IF p_tyDI.bClampRS3 = TRUE THEN
		tyP0924ClampWithRS.tyClamp3WithRSCom.tyBitmapMc.usiValueIdx	:= 1;
	ELSE
		tyP0924ClampWithRS.tyClamp3WithRSCom.tyBitmapMc.usiValueIdx	:= 0;
	END_IF

END_ACTION
```

#### Act_OptP0924Clamp3FB.st
```iecst
ACTION Act_OptP0924Clamp3FB:

	IF tyP0924ClampWithRS.tyClamp3WithRSCom.tyBtnSwitch.bValue = FALSE THEN

		IF tyP0924ClampWithRS.tyClamp3WithRSFB.tyBtnExt.bRtCompl = TRUE THEN
			tyP0924ClampWithRS.tyClamp3WithRSFB.tyBtnExt.bRtCompl	:= FALSE;

			tyP0924ClampWithRS.tyClamp3WithRSFB.tyBtnExt.bValue	:= TRUE;
			tyP0924ClampWithRS.tyClamp3WithRSFB.tyBtnRet.bValue	:= FALSE;

		ELSIF tyP0924ClampWithRS.tyClamp3WithRSFB.tyBtnRet.bRtCompl = TRUE THEN
			tyP0924ClampWithRS.tyClamp3WithRSFB.tyBtnRet.bRtCompl	:= FALSE;

			tyP0924ClampWithRS.tyClamp3WithRSFB.tyBtnRet.bValue	:= TRUE;
			tyP0924ClampWithRS.tyClamp3WithRSFB.tyBtnExt.bValue	:= FALSE;
		END_IF

		IF tyP0924ClampWithRS.tyClamp3WithRSFB.tyBtnExt.bValue = TRUE THEN
			eClamp3Act	:= PneuActExt;

			IF p_eClamp3Stat = PneuActExt AND p_eClamp3Status = Done THEN
				eClamp3Act	:= PneuActIdle;

				tyP0924ClampWithRS.tyClamp3WithRSFB.tyBtnExt.bValue	:= FALSE;

			ELSIF p_eClamp3Status = Error THEN
				tyP0924ClampWithRS.tyClamp3WithRSFB.tyBtnExt.bValue	:= FALSE;
			END_IF

		ELSIF tyP0924ClampWithRS.tyClamp3WithRSFB.tyBtnRet.bValue = TRUE THEN
			eClamp3Act	:= PneuActRet;

			IF p_eClamp3Stat = PneuActRet AND p_eClamp3Status = Done THEN
				eClamp3Act	:= PneuActIdle;

				tyP0924ClampWithRS.tyClamp3WithRSFB.tyBtnRet.bValue := FALSE;
			ELSIF p_eClamp3Status = Error THEN
				tyP0924ClampWithRS.tyClamp3WithRSFB.tyBtnRet.bValue := FALSE;
			END_IF
		END_IF

		//Update Direct Control Status
		tyP0924ClampWithRS.tyClamp3WithRSDC.tyBtnExt.bRtCompl	:= FALSE;
		tyP0924ClampWithRS.tyClamp3WithRSDC.tyBtnRet.bRtCompl	:= FALSE;
		tyP0924ClampWithRS.tyClamp3WithRSDC.tyBtnExt.bValue	:= p_bClamp3ExtCtrl;
		tyP0924ClampWithRS.tyClamp3WithRSDC.tyBtnRet.bValue	:= p_bClamp3RetCtrl;

		IF p_tyUsrMgmtCurrAccessRgt.bManualFBOnly THEN
			fUIInRtStatOff(ADR(tyP0924ClampWithRS.tyClamp3WithRSCom.tyBtnSwitch.uiMaskRtStat));
		ELSE
			fUIInRtStatHide(ADR(tyP0924ClampWithRS.tyClamp3WithRSCom.tyBtnSwitch.uiMaskRtStat));
		END_IF

	END_IF

END_ACTION
```

#### Act_OptP0924Clamp3FBStat.st
```iecst
ACTION Act_OptP0924Clamp3FBStat:

	tyP0924ClampWithRS.tyClamp3WithRSFB.tyStringStat.sValue	:= p_sClamp3StatTxt;

END_ACTION
```

#### Act_OptP0924Clamp3DC.st
```iecst
ACTION Act_OptP0924Clamp3DC:
	IF tyP0924ClampWithRS.tyClamp3WithRSCom.tyBtnSwitch.bValue = TRUE THEN
		IF p_bClamp3TwoCtrlOut = FALSE THEN
			IF tyP0924ClampWithRS.tyClamp3WithRSDC.tyBtnExt.bRtCompl = TRUE THEN
				tyP0924ClampWithRS.tyClamp3WithRSDC.tyBtnExt.bValue	:= TRUE;
				tyP0924ClampWithRS.tyClamp3WithRSDC.tyBtnRet.bValue	:= FALSE;

				eClamp3Act	:= PneuActSetExt;

				IF p_eClamp3Stat = PneuActSetExt AND p_eClamp3Status = Done THEN
					eClamp3Act	:= PneuActIdle;

					tyP0924ClampWithRS.tyClamp3WithRSDC.tyBtnExt.bRtCompl	:= FALSE;
				END_IF

			ELSIF tyP0924ClampWithRS.tyClamp3WithRSDC.tyBtnRet.bRtCompl = TRUE THEN
				tyP0924ClampWithRS.tyClamp3WithRSDC.tyBtnRet.bValue	:= TRUE;
				tyP0924ClampWithRS.tyClamp3WithRSDC.tyBtnExt.bValue	:= FALSE;

				eClamp3Act	:= PneuActSetRet;

				IF p_eClamp3Stat = PneuActSetRet AND p_eClamp3Status = Done THEN
					eClamp3Act	:= PneuActIdle;

					tyP0924ClampWithRS.tyClamp3WithRSDC.tyBtnRet.bRtCompl	:= FALSE;
				END_IF
			END_IF

		ELSE
			IF (tyP0924ClampWithRS.tyClamp3WithRSDC.tyBtnExt.bRtCompl = TRUE) OR (tyP0924ClampWithRS.tyClamp3WithRSDC.tyBtnRet.bRtCompl = TRUE) THEN
				IF (tyP0924ClampWithRS.tyClamp3WithRSDC.tyBtnExt.bValue = TRUE) AND (tyP0924ClampWithRS.tyClamp3WithRSDC.tyBtnRet.bValue = TRUE) THEN
					eClamp3Act	:= PneuActSetAll;

					IF p_eClamp3Stat = PneuActSetAll AND p_eClamp3Status = Done THEN
						eClamp3Act	:= PneuActIdle;

						tyP0924ClampWithRS.tyClamp3WithRSDC.tyBtnExt.bRtCompl	:= FALSE;
						tyP0924ClampWithRS.tyClamp3WithRSDC.tyBtnRet.bRtCompl	:= FALSE;
					END_IF

				ELSIF (tyP0924ClampWithRS.tyClamp3WithRSDC.tyBtnExt.bValue = TRUE) AND (tyP0924ClampWithRS.tyClamp3WithRSDC.tyBtnRet.bValue = FALSE) THEN
					eClamp3Act	:= PneuActSetExt;

					IF p_eClamp3Stat = PneuActSetExt AND p_eClamp3Status = Done THEN
						eClamp3Act	:= PneuActIdle;

						tyP0924ClampWithRS.tyClamp3WithRSDC.tyBtnExt.bRtCompl	:= FALSE;
						tyP0924ClampWithRS.tyClamp3WithRSDC.tyBtnRet.bRtCompl	:= FALSE;
					END_IF

				ELSIF (tyP0924ClampWithRS.tyClamp3WithRSDC.tyBtnExt.bValue = FALSE) AND (tyP0924ClampWithRS.tyClamp3WithRSDC.tyBtnRet.bValue = TRUE) THEN
					eClamp3Act	:= PneuActSetRet;

					IF p_eClamp3Stat = PneuActSetRet AND p_eClamp3Status = Done THEN
						eClamp3Act	:= PneuActIdle;

						tyP0924ClampWithRS.tyClamp3WithRSDC.tyBtnExt.bRtCompl	:= FALSE;
						tyP0924ClampWithRS.tyClamp3WithRSDC.tyBtnRet.bRtCompl	:= FALSE;
					END_IF

				ELSE
					eClamp3Act	:= PneuActRstAll;

					IF p_eClamp3Stat = PneuActRstAll AND p_eClamp3Status = Done THEN
						eClamp3Act	:= PneuActIdle;

						tyP0924ClampWithRS.tyClamp3WithRSDC.tyBtnExt.bRtCompl	:= FALSE;
						tyP0924ClampWithRS.tyClamp3WithRSDC.tyBtnRet.bRtCompl	:= FALSE;
					END_IF

				END_IF
			END_IF
		END_IF

		tyP0924ClampWithRS.tyClamp3WithRSFB.tyBtnRet.bRtCompl	:= FALSE;
		tyP0924ClampWithRS.tyClamp3WithRSFB.tyBtnRet.bValue	:= FALSE;
		tyP0924ClampWithRS.tyClamp3WithRSFB.tyBtnExt.bRtCompl	:= FALSE;
		tyP0924ClampWithRS.tyClamp3WithRSFB.tyBtnExt.bValue	:= FALSE;

	END_IF

END_ACTION
```

#### Act_OptP0924RstMnl.st
```iecst
ACTION Act_OptP0924RstMnl:

	IF EDGEPOS(p_eClamp1Status = Error) THEN

		eClamp1Act	:= PneuActIdle;

		tyP0924ClampWithRS.tyClamp1WithRSDC.tyBtnExt.bRtCompl	:= FALSE;
		tyP0924ClampWithRS.tyClamp1WithRSDC.tyBtnExt.bValue	:= FALSE;
		tyP0924ClampWithRS.tyClamp1WithRSDC.tyBtnRet.bRtCompl	:= FALSE;
		tyP0924ClampWithRS.tyClamp1WithRSDC.tyBtnRet.bValue	:= TRUE;

		tyP0924ClampWithRS.tyClamp1WithRSFB.tyBtnExt.bRtCompl	:= FALSE;
		tyP0924ClampWithRS.tyClamp1WithRSFB.tyBtnExt.bValue	:= FALSE;
		tyP0924ClampWithRS.tyClamp1WithRSFB.tyBtnRet.bRtCompl	:= FALSE;
		tyP0924ClampWithRS.tyClamp1WithRSFB.tyBtnRet.bValue	:= FALSE;

	END_IF

	IF EDGEPOS(p_eClamp2Status = Error) THEN

		eClamp2Act	:= PneuActIdle;

		tyP0924ClampWithRS.tyClamp2WithRSDC.tyBtnExt.bRtCompl		:= FALSE;
		tyP0924ClampWithRS.tyClamp2WithRSDC.tyBtnExt.bValue		:= FALSE;
		tyP0924ClampWithRS.tyClamp2WithRSDC.tyBtnRet.bRtCompl		:= FALSE;
		tyP0924ClampWithRS.tyClamp2WithRSDC.tyBtnRet.bValue		:= FALSE;

		tyP0924ClampWithRS.tyClamp2WithRSFB.tyBtnExt.bRtCompl		:= FALSE;
		tyP0924ClampWithRS.tyClamp2WithRSFB.tyBtnExt.bValue		:= FALSE;
		tyP0924ClampWithRS.tyClamp2WithRSFB.tyBtnRet.bRtCompl		:= FALSE;
		tyP0924ClampWithRS.tyClamp2WithRSFB.tyBtnRet.bValue		:= FALSE;

	END_IF

	IF EDGEPOS(p_eClamp3Status = Error) THEN

		eClamp3Act	:= PneuActIdle;

		tyP0924ClampWithRS.tyClamp3WithRSDC.tyBtnExt.bRtCompl		:= FALSE;
		tyP0924ClampWithRS.tyClamp3WithRSDC.tyBtnExt.bValue		:= FALSE;
		tyP0924ClampWithRS.tyClamp3WithRSDC.tyBtnRet.bRtCompl		:= FALSE;
		tyP0924ClampWithRS.tyClamp3WithRSDC.tyBtnRet.bValue		:= FALSE;

		tyP0924ClampWithRS.tyClamp3WithRSFB.tyBtnExt.bRtCompl		:= FALSE;
		tyP0924ClampWithRS.tyClamp3WithRSFB.tyBtnExt.bValue		:= FALSE;
		tyP0924ClampWithRS.tyClamp3WithRSFB.tyBtnRet.bRtCompl		:= FALSE;
		tyP0924ClampWithRS.tyClamp3WithRSFB.tyBtnRet.bValue		:= FALSE;

	END_IF

	IF EDGEPOS(bManualMod = FALSE) THEN

		tyP0924ClampWithRS.tyClamp1WithRSCom.tyBtnSwitch.bValue		:= FALSE;
		tyP0924ClampWithRS.tyClamp2WithRSCom.tyBtnSwitch.bValue		:= FALSE;
		tyP0924ClampWithRS.tyClamp3WithRSCom.tyBtnSwitch.bValue		:= FALSE;

		IF bUIManualMod=FALSE THEN
			fUIInRtStatHide(ADR(tyP0924ClampWithRS.tyClamp1WithRSDC.tyLyr.uiRtStat));
			fUIInRtStatOff(ADR(tyP0924ClampWithRS.tyClamp1WithRSFB.tyLyr.uiRtStat));

			fUIInRtStatHide(ADR(tyP0924ClampWithRS.tyClamp2WithRSDC.tyLyr.uiRtStat));
			fUIInRtStatOff(ADR(tyP0924ClampWithRS.tyClamp2WithRSFB.tyLyr.uiRtStat));

			fUIInRtStatHide(ADR(tyP0924ClampWithRS.tyClamp3WithRSDC.tyLyr.uiRtStat));
			fUIInRtStatOff(ADR(tyP0924ClampWithRS.tyClamp3WithRSFB.tyLyr.uiRtStat));
		END_IF

		eClamp1Act	:= PneuActIdle;

		tyP0924ClampWithRS.tyClamp1WithRSDC.tyBtnExt.bRtCompl	:= FALSE;
		tyP0924ClampWithRS.tyClamp1WithRSDC.tyBtnExt.bValue	:= FALSE;
		tyP0924ClampWithRS.tyClamp1WithRSDC.tyBtnRet.bRtCompl	:= FALSE;
		tyP0924ClampWithRS.tyClamp1WithRSDC.tyBtnRet.bValue	:= TRUE;

		tyP0924ClampWithRS.tyClamp1WithRSFB.tyBtnExt.bRtCompl	:= FALSE;
		tyP0924ClampWithRS.tyClamp1WithRSFB.tyBtnExt.bValue	:= FALSE;
		tyP0924ClampWithRS.tyClamp1WithRSFB.tyBtnRet.bRtCompl	:= FALSE;
		tyP0924ClampWithRS.tyClamp1WithRSFB.tyBtnRet.bValue	:= FALSE;

		eClamp2Act	:= PneuActIdle;

		tyP0924ClampWithRS.tyClamp2WithRSDC.tyBtnExt.bRtCompl		:= FALSE;
		tyP0924ClampWithRS.tyClamp2WithRSDC.tyBtnExt.bValue		:= FALSE;
		tyP0924ClampWithRS.tyClamp2WithRSDC.tyBtnRet.bRtCompl		:= FALSE;
		tyP0924ClampWithRS.tyClamp2WithRSDC.tyBtnRet.bValue		:= FALSE;

		tyP0924ClampWithRS.tyClamp2WithRSFB.tyBtnExt.bRtCompl		:= FALSE;
		tyP0924ClampWithRS.tyClamp2WithRSFB.tyBtnExt.bValue		:= FALSE;
		tyP0924ClampWithRS.tyClamp2WithRSFB.tyBtnRet.bRtCompl		:= FALSE;
		tyP0924ClampWithRS.tyClamp2WithRSFB.tyBtnRet.bValue		:= FALSE;

		eClamp3Act	:= PneuActIdle;

		tyP0924ClampWithRS.tyClamp3WithRSDC.tyBtnExt.bRtCompl		:= FALSE;
		tyP0924ClampWithRS.tyClamp3WithRSDC.tyBtnExt.bValue		:= FALSE;
		tyP0924ClampWithRS.tyClamp3WithRSDC.tyBtnRet.bRtCompl		:= FALSE;
		tyP0924ClampWithRS.tyClamp3WithRSDC.tyBtnRet.bValue		:= FALSE;

		tyP0924ClampWithRS.tyClamp3WithRSFB.tyBtnExt.bRtCompl		:= FALSE;
		tyP0924ClampWithRS.tyClamp3WithRSFB.tyBtnExt.bValue		:= FALSE;
		tyP0924ClampWithRS.tyClamp3WithRSFB.tyBtnRet.bRtCompl		:= FALSE;
		tyP0924ClampWithRS.tyClamp3WithRSFB.tyBtnRet.bValue		:= FALSE;

	END_IF
END_ACTION
```

#### Act_EntP0931Disp.st
```iecst
ACTION Act_EntP0931Disp:

	//Access Address
	p_tyC0003DualMask ACCESS ADR(tyP0931ConvInv.tyDualMaskHide);

	p_tyC0004Navi ACCESS ADR(tyP0931ConvInv.tyNaviBack);

	p_tyC0005Main ACCESS ADR(tyCommon.tyMain);

	p_tyC0007Notif ACCESS ADR(tyCommon.tyNotif);

	p_tyC0008MsgBox ACCESS ADR(tyP0931ConvInv.tyMsgBoxHide);

	p_tyC0009Info ACCESS ADR(tyCommon.tyInfo);

	p_tyP0931ConvCom ACCESS ADR(tyP0931ConvInv.tyConvCom);

	p_tyP0931ConvDC ACCESS ADR(tyP0931ConvInv.tyConvDC);

	p_tyP0931ConvFB ACCESS ADR(tyP0931ConvInv.tyConvFB);

	p_tyP0931InvCom ACCESS ADR(tyP0931ConvInv.tyInvCom);

	p_tyP0931InvDC ACCESS ADR(tyP0931ConvInv.tyInvDC);

	p_tyP0931InvFB ACCESS ADR(tyP0931ConvInv.tyInvFB);

	//Display
	IF tyP0931ConvInv.tyConvCom.tyBtnDCCtrl.bValue = TRUE THEN
		fUIInRtStatOff(ADR(tyP0931ConvInv.tyConvDC.tyLyr.uiRtStat));
		fUIInRtStatHide(ADR(tyP0931ConvInv.tyConvFB.tyLyr.uiRtStat));
	ELSE
		fUIInRtStatHide(ADR(tyP0931ConvInv.tyConvDC.tyLyr.uiRtStat));
		fUIInRtStatOff(ADR(tyP0931ConvInv.tyConvFB.tyLyr.uiRtStat));
	END_IF

	IF tyP0931ConvInv.tyInvCom.tyBtnDCCtrl.bValue = TRUE THEN
		fUIInRtStatOff(ADR(tyP0931ConvInv.tyInvDC.tyLyr.uiRtStat));
		fUIInRtStatHide(ADR(tyP0931ConvInv.tyInvFB.tyLyr.uiRtStat));
	ELSE
		fUIInRtStatHide(ADR(tyP0931ConvInv.tyInvDC.tyLyr.uiRtStat));
		fUIInRtStatOff(ADR(tyP0931ConvInv.tyInvFB.tyLyr.uiRtStat));
	END_IF

	//On Brake when Enter
	tyP0931ConvInv.tyInvDC.tyBtnBrake.bValue := FALSE;

END_ACTION
```

#### Act_OptP0931DualMask.st
```iecst
ACTION Act_OptP0931DualMask:

	IF eCurrPage = UIP0931ConvInv THEN

		IF p_tyDI.bEStopSig = FALSE THEN
			p_tyC0003DualMask ACCESS ADR(tyP0931ConvInv.tyDualMaskEStop);

		ELSIF p_tyDI.bCoverSWSig = FALSE THEN
			p_tyC0003DualMask ACCESS ADR(tyP0931ConvInv.tyDualMaskCWSig);

		ELSIF p_tyDI.bSafetyRlySig = FALSE THEN
			p_tyC0003DualMask ACCESS ADR(tyP0931ConvInv.tyDualMaskSafetyRly);

		ELSIF (p_tyNtParamCurr.bProjInletShutPrep AND p_tyMcParamCurr.bInShutterDis=FALSE AND p_tyDI.bInShutterCloseRS=FALSE) THEN
			IF  p_eOpsInvertCurrPos = InvertPosInvalid THEN
				p_tyC0003DualMask ACCESS ADR(tyP0931ConvInv.tyDualMaskInletNInvalid);
			ELSE
				p_tyC0003DualMask ACCESS ADR(tyP0931ConvInv.tyDualMaskInletShutterInterrupt);
			END_IF
		ELSIF (p_tyNtParamCurr.bProjOutletShutPrep AND p_tyMcParamCurr.bOutShutterDis=FALSE AND p_tyDI.bOutShutterCloseRS=FALSE) THEN
			IF  p_eOpsInvertCurrPos = InvertPosInvalid THEN
				p_tyC0003DualMask ACCESS ADR(tyP0931ConvInv.tyDualMaskOutletNInvalid);
			ELSE
				p_tyC0003DualMask ACCESS ADR(tyP0931ConvInv.tyDualMaskOutletShutterInterrupt);
			END_IF

		ELSIF (p_tyDI.bInvertHomeSen AND p_tyDI.bConvLftSen) OR (p_tyDI.bInvertRemoteSen AND p_tyDI.bConvRgtSen) THEN
			p_tyC0003DualMask ACCESS ADR(tyP0931ConvInv.tyDualMaskInvertInterrupt);

		ELSIF (p_tyDI.bInvertHomeSen AND p_tyDI.bConvRgtSen AND p_bStopperExtended = FALSE)
			OR (p_tyDI.bInvertRemoteSen AND p_tyDI.bConvLftSen AND p_bStopperExtended = FALSE)
			THEN
			p_tyC0003DualMask ACCESS ADR(tyP0931ConvInv.tyDualMaskStopperInterruptInv);

		ELSIF  p_eOpsInvertCurrPos = InvertPosInvalid THEN
			p_tyC0003DualMask ACCESS ADR(tyP0931ConvInv.tyDualMaskInvalidPos);

		ELSE
			p_tyC0003DualMask ACCESS ADR(tyP0931ConvInv.tyDualMaskHide);

		END_IF

	END_IF

END_ACTION
```

#### Act_OptP0931Navi.st
```iecst
ACTION Act_OptP0931Navi:

	IF tyP0931ConvInv.tyNaviBack.tyBtnBack.bRtCompl = TRUE THEN
		tyP0931ConvInv.tyNaviBack.tyBtnBack.bRtCompl 	:= FALSE;
		tyP0931ConvInv.tyNaviBack.tyBtnBack.bValue		:= FALSE;

		eChgPage	:= UIP0920MtrNPneuCtrl;

	END_IF

END_ACTION
```

#### Act_OptP0931Sen.st
```iecst
ACTION Act_OptP0931Sen:

	tyP0931ConvInv.tyConvCom.tyBtnLft.bValue		:= p_tyDI.bConvLftSen;
	tyP0931ConvInv.tyConvCom.tyBtnRgt.bValue		:= p_tyDI.bConvRgtSen;

	tyP0931ConvInv.tyInvCom.tyBtnHomeSen.bValue		:= p_tyDI.bInvertHomeSen;
	tyP0931ConvInv.tyInvCom.tyBtnRemoteSen.bValue	:= p_tyDI.bInvertRemoteSen;

END_ACTION
```

#### Act_OptP0931ConvChgLyr.st
```iecst
ACTION Act_OptP0931ConvChgLyr:

	IF tyP0931ConvInv.tyConvCom.tyBtnDCCtrl.bValue = TRUE THEN
		fUIInRtStatOff(ADR(tyP0931ConvInv.tyConvDC.tyLyr.uiRtStat));
		fUIInRtStatHide(ADR(tyP0931ConvInv.tyConvFB.tyLyr.uiRtStat));
	ELSE
		fUIInRtStatHide(ADR(tyP0931ConvInv.tyConvDC.tyLyr.uiRtStat));
		fUIInRtStatOff(ADR(tyP0931ConvInv.tyConvFB.tyLyr.uiRtStat));
	END_IF

END_ACTION
```

#### Act_OptP0931ConvFB.st
```iecst
ACTION Act_OptP0931ConvFB:

	IF tyP0931ConvInv.tyConvFB.tyBtnStop.bRtCompl = TRUE THEN
		eConvAct	:= ConvActStop;

		IF p_eConvStat = ConvActStop AND p_eConvStatus = Done THEN
			eConvAct	:= ConvActIdle;

			tyP0931ConvInv.tyConvFB.tyBtnEnt.bRtCompl	:= FALSE;
			tyP0931ConvInv.tyConvFB.tyBtnEnt.bValue	:= FALSE;
			tyP0931ConvInv.tyConvFB.tyBtnEnt.bRtLk		:= FALSE;

			tyP0931ConvInv.tyConvFB.tyBtnExit.bRtCompl	:= FALSE;
			tyP0931ConvInv.tyConvFB.tyBtnExit.bValue	:= FALSE;
			tyP0931ConvInv.tyConvFB.tyBtnExit.bRtLk	:= FALSE;

			tyP0931ConvInv.tyConvFB.tyBtnPreExit.bRtCompl	:= FALSE;
			tyP0931ConvInv.tyConvFB.tyBtnPreExit.bValue	:= FALSE;
			tyP0931ConvInv.tyConvFB.tyBtnPreExit.bRtLk		:= FALSE;

			tyP0931ConvInv.tyConvFB.tyBtnStop.bRtCompl	:= FALSE;
			tyP0931ConvInv.tyConvFB.tyBtnStop.bValue	:= TRUE;
			tyP0931ConvInv.tyConvFB.tyBtnStop.bRtLk	:= TRUE;

			//Unmask
			fUIInRtStatHide(ADR(tyP0931ConvInv.tyConvFB.tyBtnEnt.uiMaskRtStat));
			fUIInRtStatHide(ADR(tyP0931ConvInv.tyConvFB.tyBtnExit.uiMaskRtStat));
			fUIInRtStatHide(ADR(tyP0931ConvInv.tyConvFB.tyBtnPreExit.uiMaskRtStat));
			fUIInRtStatHide(ADR(tyP0931ConvInv.tyConvCom.tyBtnDCCtrl.uiMaskRtStat));
		END_IF

	ELSIF tyP0931ConvInv.tyConvFB.tyBtnEnt.bRtCompl = TRUE THEN
		tyP0931ConvInv.tyConvFB.tyBtnEnt.bValue	:= TRUE;
		tyP0931ConvInv.tyConvFB.tyBtnEnt.bRtLk		:= TRUE;

		tyP0931ConvInv.tyConvFB.tyBtnStop.bValue	:= FALSE;
		tyP0931ConvInv.tyConvFB.tyBtnStop.bRtLk	:= FALSE;

		IF p_eOpsInvertCurrPos = InvertCurrPosAtRemote THEN

			CASE usiConvStep OF
				0:
					eConvAct	:= ConvActEntToInOff;

					IF p_eConvStat = ConvActEntToInOff AND p_eConvStatus = Done THEN
						eConvAct	:= ConvActIdle;

						usiConvStep	:= 1;
					END_IF

				1:
					eConvAct	:= ConvActRevImmedStart;

					IF p_eConvStat = ConvActRevImmedStart AND p_eConvStatus = Done THEN
						eConvAct	:= ConvActIdle;

						usiConvStep	:= 0;

						tyP0931ConvInv.tyConvFB.tyBtnEnt.bRtCompl	:= FALSE;

						tyP0931ConvInv.tyConvFB.tyBtnEnt.bValue	:= FALSE;
						tyP0931ConvInv.tyConvFB.tyBtnEnt.bRtLk		:= FALSE;

						tyP0931ConvInv.tyConvFB.tyBtnStop.bValue	:= TRUE;
						tyP0931ConvInv.tyConvFB.tyBtnStop.bRtLk	:= TRUE;

					END_IF

			END_CASE

		ELSIF p_eOpsInvertCurrPos = InvertCurrPosAtHome THEN

			eConvAct	:= ConvActEnt;

			IF p_eConvStat = ConvActEnt AND p_eConvStatus = Done THEN
				eConvAct	:= ConvActIdle;

				tyP0931ConvInv.tyConvFB.tyBtnEnt.bRtCompl	:= FALSE;

				tyP0931ConvInv.tyConvFB.tyBtnEnt.bValue	:= FALSE;
				tyP0931ConvInv.tyConvFB.tyBtnEnt.bRtLk		:= FALSE;

				tyP0931ConvInv.tyConvFB.tyBtnStop.bValue	:= TRUE;
				tyP0931ConvInv.tyConvFB.tyBtnStop.bRtLk	:= TRUE;

			END_IF

		END_IF

	ELSIF tyP0931ConvInv.tyConvFB.tyBtnExit.bRtCompl = TRUE THEN
		tyP0931ConvInv.tyConvFB.tyBtnExit.bValue	:= TRUE;
		tyP0931ConvInv.tyConvFB.tyBtnExit.bRtLk	:= TRUE;

		tyP0931ConvInv.tyConvFB.tyBtnStop.bValue	:= FALSE;
		tyP0931ConvInv.tyConvFB.tyBtnStop.bRtLk	:= FALSE;

		eConvAct	:= ConvActExit;

		IF p_eConvStat = ConvActExit AND p_eConvStatus = Done THEN
			eConvAct	:= ConvActIdle;

			tyP0931ConvInv.tyConvFB.tyBtnExit.bRtCompl	:= FALSE;

			tyP0931ConvInv.tyConvFB.tyBtnExit.bValue	:= FALSE;
			tyP0931ConvInv.tyConvFB.tyBtnExit.bRtLk	:= FALSE;

			tyP0931ConvInv.tyConvFB.tyBtnStop.bValue	:= TRUE;
			tyP0931ConvInv.tyConvFB.tyBtnStop.bRtLk	:= TRUE;

		END_IF

	ELSIF tyP0931ConvInv.tyConvFB.tyBtnPreExit.bRtCompl = TRUE THEN
		tyP0931ConvInv.tyConvFB.tyBtnPreExit.bValue	:= TRUE;
		tyP0931ConvInv.tyConvFB.tyBtnPreExit.bRtLk		:= TRUE;

		tyP0931ConvInv.tyConvFB.tyBtnStop.bValue	:= FALSE;
		tyP0931ConvInv.tyConvFB.tyBtnStop.bRtLk	:= FALSE;

		eConvAct	:= ConvActPreExit;

		IF p_eConvStat = ConvActPreExit AND p_eConvStatus = Done THEN
			eConvAct	:= ConvActIdle;

			tyP0931ConvInv.tyConvFB.tyBtnPreExit.bRtCompl	:= FALSE;

			tyP0931ConvInv.tyConvFB.tyBtnPreExit.bValue	:= FALSE;
			tyP0931ConvInv.tyConvFB.tyBtnPreExit.bRtLk		:= FALSE;

			tyP0931ConvInv.tyConvFB.tyBtnStop.bValue		:= TRUE;
			tyP0931ConvInv.tyConvFB.tyBtnStop.bRtLk		:= TRUE;

		END_IF

	END_IF

	//Mask
	IF p_tyUsrMgmtCurrAccessRgt.bManualFBOnly THEN

		fUIInRtStatOff(ADR(tyP0931ConvInv.tyConvCom.tyBtnDCCtrl.uiMaskRtStat));

		IF (p_eConvStatus = Error) OR NOT p_tyDI.bSafetyRlySig THEN

			fUIInRtStatOff(ADR(tyP0931ConvInv.tyConvFB.tyBtnEnt.uiMaskRtStat));
			fUIInRtStatOff(ADR(tyP0931ConvInv.tyConvFB.tyBtnExit.uiMaskRtStat));
			fUIInRtStatOff(ADR(tyP0931ConvInv.tyConvFB.tyBtnPreExit.uiMaskRtStat));

		ELSIF tyP0931ConvInv.tyConvFB.tyBtnEnt.bRtCompl = TRUE THEN

			fUIInRtStatHide(ADR(tyP0931ConvInv.tyConvFB.tyBtnEnt.uiMaskRtStat));
			fUIInRtStatOff(ADR(tyP0931ConvInv.tyConvFB.tyBtnExit.uiMaskRtStat));
			fUIInRtStatOff(ADR(tyP0931ConvInv.tyConvFB.tyBtnPreExit.uiMaskRtStat));

		ELSIF tyP0931ConvInv.tyConvFB.tyBtnExit.bRtCompl = TRUE THEN

			fUIInRtStatHide(ADR(tyP0931ConvInv.tyConvFB.tyBtnExit.uiMaskRtStat));
			fUIInRtStatOff(ADR(tyP0931ConvInv.tyConvFB.tyBtnEnt.uiMaskRtStat));
			fUIInRtStatOff(ADR(tyP0931ConvInv.tyConvFB.tyBtnPreExit.uiMaskRtStat));

		ELSIF tyP0931ConvInv.tyConvFB.tyBtnPreExit.bRtCompl = TRUE THEN

			fUIInRtStatHide(ADR(tyP0931ConvInv.tyConvFB.tyBtnPreExit.uiMaskRtStat));
			fUIInRtStatOff(ADR(tyP0931ConvInv.tyConvFB.tyBtnEnt.uiMaskRtStat));
			fUIInRtStatOff(ADR(tyP0931ConvInv.tyConvFB.tyBtnExit.uiMaskRtStat));

		ELSE

			fUIInRtStatHide(ADR(tyP0931ConvInv.tyConvFB.tyBtnEnt.uiMaskRtStat));
			fUIInRtStatHide(ADR(tyP0931ConvInv.tyConvFB.tyBtnExit.uiMaskRtStat));

			IF p_eOpsInvertCurrPos=InvertCurrPosAtRemote THEN
				fUIInRtStatHide(ADR(tyP0931ConvInv.tyConvFB.tyBtnPreExit.uiMaskRtStat));
			ELSE
				fUIInRtStatOff(ADR(tyP0931ConvInv.tyConvFB.tyBtnPreExit.uiMaskRtStat));
			END_IF

		END_IF

	ELSE
		//Mask
		IF (p_eConvStatus = Error) OR NOT p_tyDI.bSafetyRlySig THEN

			fUIInRtStatOff(ADR(tyP0931ConvInv.tyConvFB.tyBtnEnt.uiMaskRtStat));
			fUIInRtStatOff(ADR(tyP0931ConvInv.tyConvFB.tyBtnExit.uiMaskRtStat));
			fUIInRtStatOff(ADR(tyP0931ConvInv.tyConvFB.tyBtnPreExit.uiMaskRtStat));
			fUIInRtStatHide(ADR(tyP0931ConvInv.tyConvCom.tyBtnDCCtrl.uiMaskRtStat));

		ELSIF tyP0931ConvInv.tyConvFB.tyBtnEnt.bRtCompl = TRUE THEN

			fUIInRtStatHide(ADR(tyP0931ConvInv.tyConvFB.tyBtnEnt.uiMaskRtStat));
			fUIInRtStatOff(ADR(tyP0931ConvInv.tyConvFB.tyBtnExit.uiMaskRtStat));
			fUIInRtStatOff(ADR(tyP0931ConvInv.tyConvFB.tyBtnPreExit.uiMaskRtStat));
			fUIInRtStatOff(ADR(tyP0931ConvInv.tyConvCom.tyBtnDCCtrl.uiMaskRtStat));

		ELSIF tyP0931ConvInv.tyConvFB.tyBtnExit.bRtCompl =TRUE THEN

			fUIInRtStatOff(ADR(tyP0931ConvInv.tyConvFB.tyBtnEnt.uiMaskRtStat));
			fUIInRtStatHide(ADR(tyP0931ConvInv.tyConvFB.tyBtnExit.uiMaskRtStat));
			fUIInRtStatOff(ADR(tyP0931ConvInv.tyConvFB.tyBtnPreExit.uiMaskRtStat));
			fUIInRtStatOff(ADR(tyP0931ConvInv.tyConvCom.tyBtnDCCtrl.uiMaskRtStat));

		ELSIF tyP0931ConvInv.tyConvFB.tyBtnPreExit.bRtCompl = TRUE THEN

			fUIInRtStatOff(ADR(tyP0931ConvInv.tyConvFB.tyBtnEnt.uiMaskRtStat));
			fUIInRtStatOff(ADR(tyP0931ConvInv.tyConvFB.tyBtnExit.uiMaskRtStat));
			fUIInRtStatHide(ADR(tyP0931ConvInv.tyConvFB.tyBtnPreExit.uiMaskRtStat));
			fUIInRtStatOff(ADR(tyP0931ConvInv.tyConvCom.tyBtnDCCtrl.uiMaskRtStat));

		ELSE
		//Unmask
			fUIInRtStatHide(ADR(tyP0931ConvInv.tyConvFB.tyBtnEnt.uiMaskRtStat));
			fUIInRtStatHide(ADR(tyP0931ConvInv.tyConvFB.tyBtnExit.uiMaskRtStat));
			fUIInRtStatHide(ADR(tyP0931ConvInv.tyConvCom.tyBtnDCCtrl.uiMaskRtStat));

			IF p_eOpsInvertCurrPos=InvertCurrPosAtRemote THEN
				fUIInRtStatHide(ADR(tyP0931ConvInv.tyConvFB.tyBtnPreExit.uiMaskRtStat));
			ELSE
				fUIInRtStatOff(ADR(tyP0931ConvInv.tyConvFB.tyBtnPreExit.uiMaskRtStat));
			END_IF

		END_IF

	END_IF

END_ACTION
```

#### Act_OptP0931ConvFBStat.st
```iecst
ACTION Act_OptP0931ConvFBStat:

	tyP0931ConvInv.tyConvFB.tyStringStat.sValue	:= p_sConvStatTxt;

END_ACTION
```

#### Act_OptP0931ConvDC.st
```iecst
ACTION Act_OptP0931ConvDC:

	IF tyP0931ConvInv.tyConvDC.tyBtnStop.bRtCompl = TRUE THEN
		tyP0931ConvInv.tyConvDC.tyBtnStop.bValue	:= TRUE;
		tyP0931ConvInv.tyConvDC.tyBtnStop.bRtLk	:= TRUE;

		tyP0931ConvInv.tyConvDC.tyBtnConvLToR.bValue	:= FALSE;
		tyP0931ConvInv.tyConvDC.tyBtnConvLToR.bRtLk	:= FALSE;

		tyP0931ConvInv.tyConvDC.tyBtnConvRToL.bValue	:= FALSE;
		tyP0931ConvInv.tyConvDC.tyBtnConvRToL.bRtLk	:= FALSE;

		fUIInRtStatHide(ADR(tyP0931ConvInv.tyConvDC.tyBtnConvLToR.uiMaskRtStat));
		fUIInRtStatHide(ADR(tyP0931ConvInv.tyConvDC.tyBtnConvRToL.uiMaskRtStat));
		fUIInRtStatHide(ADR(tyP0931ConvInv.tyConvCom.tyBtnDCCtrl.uiMaskRtStat));

		eConvAct	:= ConvActStop;

		IF p_eConvStat = ConvActStop AND p_eConvStatus = Done THEN
			eConvAct	:= ConvActIdle;

			tyP0931ConvInv.tyConvDC.tyBtnStop.bRtCompl	:= FALSE;
		END_IF

	ELSIF tyP0931ConvInv.tyConvDC.tyBtnConvLToR.bRtCompl = TRUE THEN
		tyP0931ConvInv.tyConvDC.tyBtnConvLToR.bValue	:= TRUE;
		tyP0931ConvInv.tyConvDC.tyBtnConvLToR.bRtLk		:= TRUE;

		tyP0931ConvInv.tyConvDC.tyBtnConvRToL.bValue	:= FALSE;
		tyP0931ConvInv.tyConvDC.tyBtnConvRToL.bRtLk	:= FALSE;

		tyP0931ConvInv.tyConvDC.tyBtnStop.bValue	:= FALSE;
		tyP0931ConvInv.tyConvDC.tyBtnStop.bRtLk	:= FALSE;

		fUIInRtStatOff(ADR(tyP0931ConvInv.tyConvDC.tyBtnConvRToL.uiMaskRtStat));
		fUIInRtStatOff(ADR(tyP0931ConvInv.tyConvCom.tyBtnDCCtrl.uiMaskRtStat));

		IF p_eOpsInvertCurrPos = InvertCurrPosAtRemote THEN

			eConvAct	:= ConvActSetMtrDirOrRToL;

			IF p_eConvStat = ConvActSetMtrDirOrRToL AND p_eConvStatus = Done THEN
				eConvAct	:= ConvActIdle;

				tyP0931ConvInv.tyConvDC.tyBtnConvLToR.bRtCompl	:= FALSE;
			END_IF

		ELSE
			eConvAct	:= ConvActSetMtrSigOnOrLToR;

			IF p_eConvStat = ConvActSetMtrSigOnOrLToR AND p_eConvStatus = Done THEN
				eConvAct	:= ConvActIdle;

				tyP0931ConvInv.tyConvDC.tyBtnConvLToR.bRtCompl	:= FALSE;
			END_IF
		END_IF
	ELSIF tyP0931ConvInv.tyConvDC.tyBtnConvRToL.bRtCompl = TRUE THEN
		tyP0931ConvInv.tyConvDC.tyBtnConvRToL.bValue	:= TRUE;
		tyP0931ConvInv.tyConvDC.tyBtnConvRToL.bRtLk	:= TRUE;

		tyP0931ConvInv.tyConvDC.tyBtnConvLToR.bValue	:= FALSE;
		tyP0931ConvInv.tyConvDC.tyBtnConvLToR.bRtLk		:= FALSE;

		tyP0931ConvInv.tyConvDC.tyBtnStop.bValue	:= FALSE;
		tyP0931ConvInv.tyConvDC.tyBtnStop.bRtLk	:= FALSE;

		fUIInRtStatOff(ADR(tyP0931ConvInv.tyConvDC.tyBtnConvLToR.uiMaskRtStat));
		fUIInRtStatOff(ADR(tyP0931ConvInv.tyConvCom.tyBtnDCCtrl.uiMaskRtStat));

		IF p_eOpsInvertCurrPos = InvertCurrPosAtRemote THEN
			eConvAct	:= ConvActSetMtrSigOnOrLToR;

			IF p_eConvStat = ConvActSetMtrSigOnOrLToR AND p_eConvStatus = Done THEN
				eConvAct	:= ConvActIdle;

				tyP0931ConvInv.tyConvDC.tyBtnConvRToL.bRtCompl	:= FALSE;
			END_IF

		ELSE
			eConvAct	:= ConvActSetMtrDirOrRToL;

			IF p_eConvStat = ConvActSetMtrDirOrRToL AND p_eConvStatus = Done THEN
				eConvAct	:= ConvActIdle;

				tyP0931ConvInv.tyConvDC.tyBtnConvRToL.bRtCompl	:= FALSE;
			END_IF
		END_IF
	END_IF

END_ACTION
```

#### Act_OptP0931InvChgLyr.st
```iecst
ACTION Act_OptP0931InvChgLyr:

	IF tyP0931ConvInv.tyInvCom.tyBtnDCCtrl.bValue = TRUE THEN
		fUIInRtStatOff(ADR(tyP0931ConvInv.tyInvDC.tyLyr.uiRtStat));
		fUIInRtStatHide(ADR(tyP0931ConvInv.tyInvFB.tyLyr.uiRtStat));
	ELSE
		fUIInRtStatHide(ADR(tyP0931ConvInv.tyInvDC.tyLyr.uiRtStat));
		fUIInRtStatOff(ADR(tyP0931ConvInv.tyInvFB.tyLyr.uiRtStat));
	END_IF

END_ACTION
```

#### Act_OptP0931InvUpdtData.st
```iecst
ACTION Act_OptP0931InvUpdtData:

	//Machine Bitmap
	IF p_tyDI.bInvertHomeSen THEN
		IF p_tyNtParamCurr.tyDOSettings.diTLGreen<>0 OR p_tyNtParamCurr.tyDOSettings.diTLAmber<>0 OR p_tyNtParamCurr.tyDOSettings.diTLRed<>0 THEN
			IF p_tyNtParamCurr.eTLBuzMode=TLBuzModBHTC THEN
				tyP0931ConvInv.tyInvCom.tyBitmapMc.usiValueIdx	:= 200;
			ELSE
				tyP0931ConvInv.tyInvCom.tyBitmapMc.usiValueIdx	:= 100;
			END_IF
		ELSE
			tyP0931ConvInv.tyInvCom.tyBitmapMc.usiValueIdx	:= 0;
		END_IF
	ELSE
		IF p_tyNtParamCurr.tyDOSettings.diTLGreen<>0 OR p_tyNtParamCurr.tyDOSettings.diTLAmber<>0 OR p_tyNtParamCurr.tyDOSettings.diTLRed<>0 THEN
			IF p_tyNtParamCurr.eTLBuzMode=TLBuzModBHTC THEN
				tyP0931ConvInv.tyInvCom.tyBitmapMc.usiValueIdx	:= 201;
			ELSE
				tyP0931ConvInv.tyInvCom.tyBitmapMc.usiValueIdx	:= 101;
			END_IF
		ELSE
			tyP0931ConvInv.tyInvCom.tyBitmapMc.usiValueIdx	:= 1;
		END_IF
	END_IF

END_ACTION
```

#### Act_OptP0931InvDC.st
```iecst
ACTION Act_OptP0931InvDC:

	IF tyP0931ConvInv.tyInvDC.tyBtnBrake.bRtCompl = TRUE THEN

		IF tyP0931ConvInv.tyInvDC.tyBtnBrake.bValue = TRUE THEN
			eInvertAct	:= MotorBrkActSetMtrBrkRls;

			IF p_eInvertStat = MotorBrkActSetMtrBrkRls AND p_eInvertStatus = Done THEN
				eInvertAct	:= MotorBrkActIdle;

				tyP0931ConvInv.tyInvDC.tyBtnBrake.bRtCompl	:= FALSE;

			END_IF

		ELSE
			eInvertAct:= MotorBrkActRstMtrBrkRls;

			IF p_eInvertStat = MotorBrkActRstMtrBrkRls AND p_eInvertStatus = Done THEN
				eInvertAct	:= MotorBrkActIdle;

				tyP0931ConvInv.tyInvDC.tyBtnBrake.bRtCompl	:= FALSE;

			END_IF

		END_IF

	END_IF

	//Turn Clockwise
	IF EDGEPOS(tyP0931ConvInv.tyInvDC.tyBtnCW.bValue = TRUE) THEN
		eInvertAct	:= MotorBrkActSetMtrSigOnOrCW;

	ELSIF tyP0931ConvInv.tyInvDC.tyBtnCW.bRtCompl = TRUE THEN
		eInvertAct	:= MotorBrkActRstMtrSigOnOrCW;

		IF p_eInvertStat = MotorBrkActRstMtrSigOnOrCW AND p_eInvertStatus = Done THEN
			eInvertAct	:= MotorBrkActIdle;

			tyP0931ConvInv.tyInvDC.tyBtnCW.bRtCompl	:= FALSE;
		END_IF
	END_IF

	IF p_eInvertStat = MotorBrkActSetMtrSigOnOrCW AND p_eInvertStatus = Done THEN
		eInvertAct	:= MotorBrkActIdle;
	END_IF

	//Turn Counter-clockwise
	IF EDGEPOS(tyP0931ConvInv.tyInvDC.tyBtnCCW.bValue = TRUE) THEN
		eInvertAct	:= MotorBrkActSetMtrDirOrCCW;

	ELSIF tyP0931ConvInv.tyInvDC.tyBtnCCW.bRtCompl = TRUE THEN
		eInvertAct	:= MotorBrkActRstMtrDirOrCCW;

		IF p_eInvertStat = MotorBrkActRstMtrDirOrCCW AND p_eInvertStatus = Done THEN
			eInvertAct	:= MotorBrkActIdle;

			tyP0931ConvInv.tyInvDC.tyBtnCCW.bRtCompl	:= FALSE;
		END_IF
	END_IF

	IF p_eInvertStat = MotorBrkActSetMtrDirOrCCW AND p_eInvertStatus = Done THEN
		eInvertAct	:= MotorBrkActIdle;
	END_IF

	//Mask and Unmask condition

	IF tyP0931ConvInv.tyInvDC.tyBtnCW.bValue THEN
		fUIInRtStatOff(ADR(tyP0931ConvInv.tyInvDC.tyBtnCCW.uiMaskRtStat));
	ELSE
		fUIInRtStatHide(ADR(tyP0931ConvInv.tyInvDC.tyBtnCCW.uiMaskRtStat));
	END_IF

	IF tyP0931ConvInv.tyInvDC.tyBtnCCW.bValue THEN
		fUIInRtStatOff(ADR(tyP0931ConvInv.tyInvDC.tyBtnCW.uiMaskRtStat));
	ELSE
		fUIInRtStatHide(ADR(tyP0931ConvInv.tyInvDC.tyBtnCW.uiMaskRtStat));
	END_IF

	//Mask CW and CCW when Brake is On
	IF (tyP0931ConvInv.tyInvDC.tyBtnBrake.bValue=FALSE) THEN
		fUIInRtStatOff(ADR(tyP0931ConvInv.tyInvDC.tyBtnCW.uiMaskRtStat));
		fUIInRtStatOff(ADR(tyP0931ConvInv.tyInvDC.tyBtnCCW.uiMaskRtStat));
	ELSE
		fUIInRtStatHide(ADR(tyP0931ConvInv.tyInvDC.tyBtnCW.uiMaskRtStat));
		fUIInRtStatHide(ADR(tyP0931ConvInv.tyInvDC.tyBtnCCW.uiMaskRtStat));
	END_IF

END_ACTION
```

#### Act_OptP0931InvFB.st
```iecst
ACTION Act_OptP0931InvFB:

	IF tyP0931ConvInv.tyInvFB.tyBtnStop.bRtCompl = TRUE THEN
		eInvertAct	:= MotorBrkActStop;

		IF p_eInvertStat = MotorBrkActStop AND p_eInvertStatus = Done THEN
			eInvertAct	:= MotorBrkActIdle;

			tyP0931ConvInv.tyInvFB.tyBtnCW.bRtCompl	:= FALSE;
			tyP0931ConvInv.tyInvFB.tyBtnCW.bValue		:= FALSE;
			tyP0931ConvInv.tyInvFB.tyBtnCW.bRtLk		:= FALSE;

			tyP0931ConvInv.tyInvFB.tyBtnCCW.bRtCompl	:= FALSE;
			tyP0931ConvInv.tyInvFB.tyBtnCCW.bValue		:= FALSE;
			tyP0931ConvInv.tyInvFB.tyBtnCCW.bRtLk		:= FALSE;

			tyP0931ConvInv.tyInvDC.tyBtnBrake.bValue 	:= FALSE;

			tyP0931ConvInv.tyInvFB.tyBtnStop.bRtCompl	:= FALSE;
			tyP0931ConvInv.tyInvFB.tyBtnStop.bValue	:= TRUE;
			tyP0931ConvInv.tyInvFB.tyBtnStop.bRtLk		:= TRUE;

		END_IF

	ELSIF tyP0931ConvInv.tyInvFB.tyBtnCW.bRtCompl = TRUE THEN
		tyP0931ConvInv.tyInvFB.tyBtnCW.bValue		:= TRUE;
		tyP0931ConvInv.tyInvFB.tyBtnCW.bRtLk		:= TRUE;

		tyP0931ConvInv.tyInvFB.tyBtnStop.bValue	:= FALSE;
		tyP0931ConvInv.tyInvFB.tyBtnStop.bRtLk		:= FALSE;

		eInvertAct	:= MotorBrkActCW;

		IF p_eInvertStat = MotorBrkActCW AND p_eInvertStatus = Done THEN
			eInvertAct	:= MotorBrkActIdle;

			tyP0931ConvInv.tyInvFB.tyBtnCW.bRtCompl	:= FALSE;

			tyP0931ConvInv.tyInvFB.tyBtnCW.bValue		:= FALSE;
			tyP0931ConvInv.tyInvFB.tyBtnCW.bRtLk		:= FALSE;

			tyP0931ConvInv.tyInvDC.tyBtnBrake.bValue 	:= FALSE;

			tyP0931ConvInv.tyInvFB.tyBtnStop.bValue	:= TRUE;
			tyP0931ConvInv.tyInvFB.tyBtnStop.bRtLk		:= TRUE;

		END_IF

	ELSIF tyP0931ConvInv.tyInvFB.tyBtnCCW.bRtCompl = TRUE THEN
		tyP0931ConvInv.tyInvFB.tyBtnCCW.bValue		:= TRUE;
		tyP0931ConvInv.tyInvFB.tyBtnCCW.bRtLk		:= TRUE;

		tyP0931ConvInv.tyInvFB.tyBtnStop.bValue	:= FALSE;
		tyP0931ConvInv.tyInvFB.tyBtnStop.bRtLk		:= FALSE;

		eInvertAct	:= MotorBrkActCCW;

		IF p_eInvertStat = MotorBrkActCCW AND p_eInvertStatus = Done THEN
			eInvertAct	:= MotorBrkActIdle;

			tyP0931ConvInv.tyInvFB.tyBtnCCW.bRtCompl	:= FALSE;

			tyP0931ConvInv.tyInvFB.tyBtnCCW.bValue		:= FALSE;
			tyP0931ConvInv.tyInvFB.tyBtnCCW.bRtLk		:= FALSE;

			tyP0931ConvInv.tyInvDC.tyBtnBrake.bValue 	:= FALSE;

			tyP0931ConvInv.tyInvFB.tyBtnStop.bValue	:= TRUE;
			tyP0931ConvInv.tyInvFB.tyBtnStop.bRtLk		:= TRUE;

		END_IF

	END_IF

	//Mask
	tyP0931ConvInv.tyInvFB.tyBtnCW.uiMaskRtStat.0		:= NOT( p_eInvertStatus = Error OR tyP0931ConvInv.tyInvFB.tyBtnCCW.bRtCompl);
	tyP0931ConvInv.tyInvFB.tyBtnCCW.uiMaskRtStat.0		:= NOT( p_eInvertStatus = Error OR tyP0931ConvInv.tyInvFB.tyBtnCW.bRtCompl);

	IF p_tyUsrMgmtCurrAccessRgt.bManualFBOnly THEN

		fUIInRtStatOff(ADR(tyP0931ConvInv.tyInvCom.tyBtnDCCtrl.uiMaskRtStat));

		IF (p_eInvertStatus = Error) OR NOT p_tyDI.bSafetyRlySig THEN

			fUIInRtStatOff(ADR(tyP0931ConvInv.tyInvFB.tyBtnCW.uiMaskRtStat));
			fUIInRtStatOff(ADR(tyP0931ConvInv.tyInvFB.tyBtnCCW.uiMaskRtStat));

		ELSIF tyP0931ConvInv.tyInvFB.tyBtnCW.bRtCompl = TRUE THEN

			fUIInRtStatHide(ADR(tyP0931ConvInv.tyInvFB.tyBtnCW.uiMaskRtStat));
			fUIInRtStatOff(ADR(tyP0931ConvInv.tyInvFB.tyBtnCCW.uiMaskRtStat));

		ELSIF tyP0931ConvInv.tyInvFB.tyBtnCCW.bRtCompl =TRUE THEN

			fUIInRtStatHide(ADR(tyP0931ConvInv.tyInvFB.tyBtnCCW.uiMaskRtStat));
			fUIInRtStatOff(ADR(tyP0931ConvInv.tyInvFB.tyBtnCW.uiMaskRtStat));

		ELSE

			fUIInRtStatHide(ADR(tyP0931ConvInv.tyInvFB.tyBtnCCW.uiMaskRtStat));
			fUIInRtStatHide(ADR(tyP0931ConvInv.tyInvFB.tyBtnCW.uiMaskRtStat));

		END_IF

	ELSE
		//Mask
		IF (p_eInvertStatus = Error) OR NOT p_tyDI.bSafetyRlySig THEN

			fUIInRtStatOff(ADR(tyP0931ConvInv.tyInvFB.tyBtnCW.uiMaskRtStat));
			fUIInRtStatOff(ADR(tyP0931ConvInv.tyInvFB.tyBtnCCW.uiMaskRtStat));

		ELSIF tyP0931ConvInv.tyInvFB.tyBtnCW.bRtCompl = TRUE THEN

			fUIInRtStatHide(ADR(tyP0931ConvInv.tyInvFB.tyBtnCW.uiMaskRtStat));
			fUIInRtStatOff(ADR(tyP0931ConvInv.tyInvFB.tyBtnCCW.uiMaskRtStat));
			fUIInRtStatOff(ADR(tyP0931ConvInv.tyInvCom.tyBtnDCCtrl.uiMaskRtStat));

		ELSIF tyP0931ConvInv.tyInvFB.tyBtnCCW.bRtCompl =TRUE THEN

			fUIInRtStatHide(ADR(tyP0931ConvInv.tyInvFB.tyBtnCCW.uiMaskRtStat));
			fUIInRtStatOff(ADR(tyP0931ConvInv.tyInvFB.tyBtnCW.uiMaskRtStat));
			fUIInRtStatOff(ADR(tyP0931ConvInv.tyInvCom.tyBtnDCCtrl.uiMaskRtStat));

		ELSE

			fUIInRtStatHide(ADR(tyP0931ConvInv.tyInvFB.tyBtnCCW.uiMaskRtStat));
			fUIInRtStatHide(ADR(tyP0931ConvInv.tyInvFB.tyBtnCW.uiMaskRtStat));
			fUIInRtStatHide(ADR(tyP0931ConvInv.tyInvCom.tyBtnDCCtrl.uiMaskRtStat));

		END_IF

	END_IF

END_ACTION
```

#### Act_OptP0931InvFBStat.st
```iecst
ACTION Act_OptP0931InvFBStat:

	//Inverter
	tyP0931ConvInv.tyInvFB.tyStringStat.sValue	:= p_sInvertStatTxt;

END_ACTION
```

#### Act_OptP0931RstMnl.st
```iecst
ACTION Act_OptP0931RstMnl:

	//Conveyor
	IF EDGEPOS(p_eConvStatus = Error) THEN

		eConvAct	:= ConvActIdle;

		usiConvStep	:= 0;

		//FB
		tyP0931ConvInv.tyConvFB.tyBtnEnt.bRtCompl				:= FALSE;
		tyP0931ConvInv.tyConvFB.tyBtnExit.bRtCompl				:= FALSE;
		tyP0931ConvInv.tyConvFB.tyBtnPreExit.bRtCompl			:= FALSE;
		tyP0931ConvInv.tyConvFB.tyBtnStop.bRtCompl				:= FALSE;

		tyP0931ConvInv.tyConvFB.tyBtnEnt.bValue					:= FALSE;
		tyP0931ConvInv.tyConvFB.tyBtnExit.bValue				:= FALSE;
		tyP0931ConvInv.tyConvFB.tyBtnPreExit.bValue				:= FALSE;
		tyP0931ConvInv.tyConvFB.tyBtnStop.bValue				:= TRUE;

		tyP0931ConvInv.tyConvFB.tyBtnEnt.bRtLk					:= FALSE;
		tyP0931ConvInv.tyConvFB.tyBtnExit.bRtLk					:= FALSE;
		tyP0931ConvInv.tyConvFB.tyBtnPreExit.bRtLk				:= FALSE;
		tyP0931ConvInv.tyConvFB.tyBtnStop.bRtLk					:= TRUE;

		tyP0931ConvInv.tyConvFB.tyBtnEnt.uiMaskRtStat.0			:= TRUE;
		tyP0931ConvInv.tyConvFB.tyBtnExit.uiMaskRtStat.0		:= TRUE;
		tyP0931ConvInv.tyConvFB.tyBtnPreExit.uiMaskRtStat.0		:= TRUE;
		tyP0931ConvInv.tyConvCom.tyBtnDCCtrl.uiMaskRtStat.0		:= TRUE;

		//Direct
		tyP0931ConvInv.tyConvDC.tyBtnConvLToR.bRtCompl			:= FALSE;
		tyP0931ConvInv.tyConvDC.tyBtnConvRToL.bRtCompl			:= FALSE;
		tyP0931ConvInv.tyConvDC.tyBtnStop.bRtCompl				:= FALSE;

		tyP0931ConvInv.tyConvDC.tyBtnConvLToR.bValue			:= FALSE;
		tyP0931ConvInv.tyConvDC.tyBtnConvRToL.bValue			:= FALSE;
		tyP0931ConvInv.tyConvDC.tyBtnStop.bValue				:= TRUE;

		tyP0931ConvInv.tyConvDC.tyBtnConvLToR.bRtLk				:= FALSE;
		tyP0931ConvInv.tyConvDC.tyBtnConvRToL.bRtLk				:= FALSE;
		tyP0931ConvInv.tyConvDC.tyBtnStop.bRtLk					:= TRUE;

		tyP0931ConvInv.tyConvDC.tyBtnConvLToR.uiMaskRtStat.0	:= TRUE;
		tyP0931ConvInv.tyConvDC.tyBtnConvRToL.uiMaskRtStat.0	:= TRUE;
		tyP0931ConvInv.tyConvCom.tyBtnDCCtrl.uiMaskRtStat.0		:= TRUE;

	END_IF

	IF EDGEPOS(p_eInvertStatus = Error) THEN

		eInvertAct	:= MotorBrkActIdle;

		//Inverter FB
		tyP0931ConvInv.tyInvFB.tyBtnCW.bRtCompl					:= FALSE;
		tyP0931ConvInv.tyInvFB.tyBtnCCW.bRtCompl				:= FALSE;
		tyP0931ConvInv.tyInvFB.tyBtnStop.bRtCompl				:= FALSE;

		tyP0931ConvInv.tyInvFB.tyBtnCW.bValue					:= FALSE;
		tyP0931ConvInv.tyInvFB.tyBtnCCW.bValue					:= FALSE;
		tyP0931ConvInv.tyInvFB.tyBtnStop.bValue					:= TRUE;

		tyP0931ConvInv.tyInvFB.tyBtnCW.bRtLk					:= FALSE;
		tyP0931ConvInv.tyInvFB.tyBtnCCW.bRtLk					:= FALSE;
		tyP0931ConvInv.tyInvFB.tyBtnStop.bRtLk					:= TRUE;

		tyP0931ConvInv.tyInvFB.tyBtnCW.uiMaskRtStat.0			:= TRUE;
		tyP0931ConvInv.tyInvFB.tyBtnCCW.uiMaskRtStat.0			:= TRUE;
		tyP0931ConvInv.tyInvCom.tyBtnDCCtrl.uiMaskRtStat.0		:= TRUE;

		//Inverter Direct
		tyP0931ConvInv.tyInvDC.tyBtnCW.bRtCompl					:= FALSE;
		tyP0931ConvInv.tyInvDC.tyBtnCCW.bRtCompl				:= FALSE;
		tyP0931ConvInv.tyInvDC.tyBtnBrake.bRtCompl				:= FALSE;

		tyP0931ConvInv.tyInvDC.tyBtnCW.bValue					:= FALSE;
		tyP0931ConvInv.tyInvDC.tyBtnCCW.bValue					:= FALSE;
		tyP0931ConvInv.tyInvDC.tyBtnBrake.bValue				:= TRUE;

		tyP0931ConvInv.tyInvDC.tyBtnCW.bRtLk					:= FALSE;
		tyP0931ConvInv.tyInvDC.tyBtnCCW.bRtLk					:= FALSE;
		tyP0931ConvInv.tyInvDC.tyBtnBrake.bRtLk					:= TRUE;

		tyP0931ConvInv.tyInvDC.tyBtnCW.uiMaskRtStat.0			:= TRUE;
		tyP0931ConvInv.tyInvDC.tyBtnCCW.uiMaskRtStat.0			:= TRUE;
		tyP0931ConvInv.tyInvDC.tyBtnBrake.uiMaskRtStat.0		:= TRUE;
		tyP0931ConvInv.tyInvCom.tyBtnDCCtrl.uiMaskRtStat.0		:= TRUE;

	END_IF

	IF EDGEPOS(bManualMod = FALSE) THEN
		tyP0931ConvInv.tyConvCom.tyBtnDCCtrl.bValue := FALSE;

		fUIInRtStatHide(ADR(tyP0931ConvInv.tyConvDC.tyLyr.uiRtStat));
		fUIInRtStatOff(ADR(tyP0931ConvInv.tyConvFB.tyLyr.uiRtStat));

		tyP0931ConvInv.tyInvCom.tyBtnDCCtrl.bValue := FALSE;

		fUIInRtStatHide(ADR(tyP0931ConvInv.tyInvDC.tyLyr.uiRtStat));
		fUIInRtStatOff(ADR(tyP0931ConvInv.tyInvFB.tyLyr.uiRtStat));

		eConvAct	:= ConvActIdle;

		usiConvStep	:= 0;

		//FB
		tyP0931ConvInv.tyConvFB.tyBtnEnt.bRtCompl				:= FALSE;
		tyP0931ConvInv.tyConvFB.tyBtnExit.bRtCompl				:= FALSE;
		tyP0931ConvInv.tyConvFB.tyBtnPreExit.bRtCompl			:= FALSE;
		tyP0931ConvInv.tyConvFB.tyBtnStop.bRtCompl				:= FALSE;

		tyP0931ConvInv.tyConvFB.tyBtnEnt.bValue					:= FALSE;
		tyP0931ConvInv.tyConvFB.tyBtnExit.bValue				:= FALSE;
		tyP0931ConvInv.tyConvFB.tyBtnPreExit.bValue				:= FALSE;
		tyP0931ConvInv.tyConvFB.tyBtnStop.bValue				:= TRUE;

		tyP0931ConvInv.tyConvFB.tyBtnEnt.bRtLk					:= FALSE;
		tyP0931ConvInv.tyConvFB.tyBtnExit.bRtLk					:= FALSE;
		tyP0931ConvInv.tyConvFB.tyBtnPreExit.bRtLk				:= FALSE;
		tyP0931ConvInv.tyConvFB.tyBtnStop.bRtLk					:= TRUE;

		tyP0931ConvInv.tyConvFB.tyBtnEnt.uiMaskRtStat.0			:= TRUE;
		tyP0931ConvInv.tyConvFB.tyBtnExit.uiMaskRtStat.0		:= TRUE;
		tyP0931ConvInv.tyConvFB.tyBtnPreExit.uiMaskRtStat.0		:= TRUE;
		tyP0931ConvInv.tyConvCom.tyBtnDCCtrl.uiMaskRtStat.0		:= TRUE;

		//Direct
		tyP0931ConvInv.tyConvDC.tyBtnConvLToR.bRtCompl			:= FALSE;
		tyP0931ConvInv.tyConvDC.tyBtnConvRToL.bRtCompl			:= FALSE;
		tyP0931ConvInv.tyConvDC.tyBtnStop.bRtCompl				:= FALSE;

		tyP0931ConvInv.tyConvDC.tyBtnConvLToR.bValue			:= FALSE;
		tyP0931ConvInv.tyConvDC.tyBtnConvRToL.bValue			:= FALSE;
		tyP0931ConvInv.tyConvDC.tyBtnStop.bValue				:= TRUE;

		tyP0931ConvInv.tyConvDC.tyBtnConvLToR.bRtLk				:= FALSE;
		tyP0931ConvInv.tyConvDC.tyBtnConvRToL.bRtLk				:= FALSE;
		tyP0931ConvInv.tyConvDC.tyBtnStop.bRtLk					:= TRUE;

		tyP0931ConvInv.tyConvDC.tyBtnConvLToR.uiMaskRtStat.0	:= TRUE;
		tyP0931ConvInv.tyConvDC.tyBtnConvRToL.uiMaskRtStat.0	:= TRUE;
		tyP0931ConvInv.tyConvCom.tyBtnDCCtrl.uiMaskRtStat.0		:= TRUE;

		eInvertAct	:= MotorBrkActIdle;

		//Inverter FB
		tyP0931ConvInv.tyInvFB.tyBtnCW.bRtCompl					:= FALSE;
		tyP0931ConvInv.tyInvFB.tyBtnCCW.bRtCompl				:= FALSE;
		tyP0931ConvInv.tyInvFB.tyBtnStop.bRtCompl				:= FALSE;

		tyP0931ConvInv.tyInvFB.tyBtnCW.bValue					:= FALSE;
		tyP0931ConvInv.tyInvFB.tyBtnCCW.bValue					:= FALSE;
		tyP0931ConvInv.tyInvFB.tyBtnStop.bValue					:= TRUE;

		tyP0931ConvInv.tyInvFB.tyBtnCW.bRtLk					:= FALSE;
		tyP0931ConvInv.tyInvFB.tyBtnCCW.bRtLk					:= FALSE;
		tyP0931ConvInv.tyInvFB.tyBtnStop.bRtLk					:= TRUE;

		tyP0931ConvInv.tyInvFB.tyBtnCW.uiMaskRtStat.0			:= TRUE;
		tyP0931ConvInv.tyInvFB.tyBtnCCW.uiMaskRtStat.0			:= TRUE;
		tyP0931ConvInv.tyInvCom.tyBtnDCCtrl.uiMaskRtStat.0		:= TRUE;

		//Inverter Direct
		tyP0931ConvInv.tyInvDC.tyBtnCW.bRtCompl					:= FALSE;
		tyP0931ConvInv.tyInvDC.tyBtnCCW.bRtCompl				:= FALSE;
		tyP0931ConvInv.tyInvDC.tyBtnBrake.bRtCompl				:= FALSE;

		tyP0931ConvInv.tyInvDC.tyBtnCW.bValue					:= FALSE;
		tyP0931ConvInv.tyInvDC.tyBtnCCW.bValue					:= FALSE;
		tyP0931ConvInv.tyInvDC.tyBtnBrake.bValue				:= TRUE;

		tyP0931ConvInv.tyInvDC.tyBtnCW.bRtLk					:= FALSE;
		tyP0931ConvInv.tyInvDC.tyBtnCCW.bRtLk					:= FALSE;
		tyP0931ConvInv.tyInvDC.tyBtnBrake.bRtLk					:= TRUE;

		tyP0931ConvInv.tyInvDC.tyBtnCW.uiMaskRtStat.0			:= TRUE;
		tyP0931ConvInv.tyInvDC.tyBtnCCW.uiMaskRtStat.0			:= TRUE;
		tyP0931ConvInv.tyInvDC.tyBtnBrake.uiMaskRtStat.0		:= TRUE;
		tyP0931ConvInv.tyInvCom.tyBtnDCCtrl.uiMaskRtStat.0		:= TRUE;

	END_IF

END_ACTION
```

#### Act_EntP0934Disp.st
```iecst
ACTION Act_EntP0934Disp:

	//Access Address
	p_tyC0001MotionStd ACCESS ADR(tyP0934AW.tyMotionStd);

	p_tyC0002FullMask ACCESS ADR(tyP0934AW.tyFullMaskHide);

	p_tyC0004Navi ACCESS ADR(tyP0934AW.tyNaviBack);

	p_tyC0005Main ACCESS ADR(tyCommon.tyMain);

	p_tyC0007Notif ACCESS ADR(tyCommon.tyNotif);

	p_tyC0008MsgBox ACCESS ADR(tyP0934AW.tyMsgBoxHide);

	p_tyC0009Info ACCESS ADR(tyCommon.tyInfo);

	p_tyC0011Loading ACCESS ADR(tyCommon.tyLoading);

	p_tyP0934AW ACCESS ADR(tyP0934AW.tyAW);

	//Display
	tyP0934AW.tyAW.tyNumNewWidth.diValue	:= p_tyProdRcpCurrRcp0.diWidthInUM;

	tyP0934AW.tyMotionStd.tyBtnPwr.bValue	:= p_bAWOpenPwrOn;

	fbLmtRstTm(IN := FALSE);

END_ACTION
```

#### Act_OptP0934FullMask.st
```iecst
ACTION Act_OptP0934FullMask:

	IF eCurrPage = UIP0934AW THEN

		IF p_tyDI.bEStopSig = FALSE THEN
			p_tyC0002FullMask ACCESS ADR(tyP0934AW.tyFullMaskEStop);

		ELSIF p_tyDI.bCoverSWSig = FALSE THEN
			p_tyC0002FullMask ACCESS ADR(tyP0934AW.tyFullMaskCWSig);

		ELSIF p_tyDI.bSafetyRlySig = FALSE THEN
			p_tyC0002FullMask ACCESS ADR(tyP0934AW.tyFullMaskSafetyRly);

		ELSIF p_tyDI.bConvLftSen = TRUE THEN
			p_tyC0002FullMask ACCESS ADR(tyP0934AW.tyFullMaskLftSenInterrupt);

		ELSIF p_tyDI.bConvRgtSen = TRUE THEN
			p_tyC0002FullMask ACCESS ADR(tyP0934AW.tyFullMaskRgtSenInterrupt);

		ELSIF (p_tyNtParamCurr.bProjInletShutPrep AND p_tyMcParamCurr.bInShutterDis=FALSE AND p_tyDI.bInShutterCloseRS=FALSE) THEN
			p_tyC0002FullMask ACCESS ADR(tyP0934AW.tyFullMaskInletShutterInterrupt);

		ELSIF (p_tyNtParamCurr.bProjOutletShutPrep AND p_tyMcParamCurr.bOutShutterDis=FALSE AND p_tyDI.bOutShutterCloseRS=FALSE) THEN
			p_tyC0002FullMask ACCESS ADR(tyP0934AW.tyFullMaskOutletShutterInterrupt);

		ELSIF p_tyDI.bInvertHomeSen = FALSE AND p_tyDI.bInvertRemoteSen = FALSE THEN
			p_tyC0002FullMask ACCESS ADR(tyP0934AW.tyFullMaskHomeSenInterrupt);

		ELSE
			p_tyC0002FullMask ACCESS ADR(tyP0934AW.tyFullMaskHide);

		END_IF

	END_IF

END_ACTION
```

#### Act_OptP0934Navi.st
```iecst
ACTION Act_OptP0934Navi:

	IF tyP0934AW.tyNaviBack.tyBtnBack.bRtCompl = TRUE THEN
		tyP0934AW.tyNaviBack.tyBtnBack.bRtCompl	:= FALSE;
		tyP0934AW.tyNaviBack.tyBtnBack.bValue	:= FALSE;

		eChgPage	:= UIP0920MtrNPneuCtrl;

	END_IF

END_ACTION
```

#### Act_OptP0934FB.st
```iecst
ACTION Act_OptP0934FB:

	fbJogSlowToFastDlyTm.PT	:= T#2s;
	fbJogSlowToFastDlyTm;
	fbLmtRstTm;

	IF EDGEPOS((p_bAWOpenFwdLmtSen OR p_bAWOpenRevLmtSen OR p_udiAWOpenAxisErrID = 21570 OR p_udiAWOpenAxisErrID = 21571)
		AND tyP0934AW.tyMotionStd.tyBtnJogOpen.bValue = FALSE AND tyP0934AW.tyMotionStd.tyBtnJogClose.bValue = FALSE) THEN

		fbLmtRstTm.IN	:= TRUE;

	END_IF

	IF fbLmtRstTm.Q = TRUE THEN
		tyP0934AW.tyMotionStd.tyBtnRst.bRtCompl	:= TRUE;
	END_IF

	IF (tyP0934AW.tyMotionStd.tyBtnJogOpen.bValue = FALSE AND tyP0934AW.tyMotionStd.tyBtnJogClose.bValue = FALSE) AND (p_bAWOpenJogging = TRUE) THEN
		bJogStopAW	:= TRUE;
	END_IF

	IF tyP0934AW.tyMotionStd.tyBtnStop.bRtCompl = TRUE THEN
		eAWOpenAct		:= AWActStop;

		IF p_eAWOpenStat = AWActStop AND p_eAWOpenStatus = Done THEN
			eAWOpenAct	:= AWActIdle;

			tyP0934AW.tyMotionStd.tyBtnStop.bRtCompl			:= FALSE;
			tyP0934AW.tyMotionStd.tyBtnJogOpen.bRtCompl			:= FALSE;
			tyP0934AW.tyMotionStd.tyBtnJogClose.bRtCompl		:= FALSE;
			tyP0934AW.tyMotionStd.tyBtnOrigin.bRtCompl			:= FALSE;
			tyP0934AW.tyMotionStd.tyBtnMovAbs.bRtCompl			:= FALSE;
			tyP0934AW.tyMotionStd.tyBtnMovRel.bRtCompl			:= FALSE;
			tyP0934AW.tyAW.tyBtnGo.bRtCompl						:= FALSE;

			tyP0934AW.tyMotionStd.tyBtnStop.bValue				:= TRUE;
			tyP0934AW.tyMotionStd.tyBtnJogOpen.bValue			:= FALSE;
			tyP0934AW.tyMotionStd.tyBtnJogClose.bValue			:= FALSE;
			tyP0934AW.tyMotionStd.tyBtnOrigin.bValue			:= FALSE;
			tyP0934AW.tyMotionStd.tyBtnMovAbs.bValue			:= FALSE;
			tyP0934AW.tyMotionStd.tyBtnMovRel.bValue			:= FALSE;
			tyP0934AW.tyAW.tyBtnGo.bValue						:= FALSE;

			tyP0934AW.tyMotionStd.tyBtnStop.bRtLk				:= TRUE;
			tyP0934AW.tyMotionStd.tyBtnJogOpen.bRtLk			:= FALSE;
			tyP0934AW.tyMotionStd.tyBtnJogClose.bRtLk			:= FALSE;
			tyP0934AW.tyMotionStd.tyBtnOrigin.bRtLk				:= FALSE;
			tyP0934AW.tyMotionStd.tyBtnMovAbs.bRtLk				:= FALSE;
			tyP0934AW.tyMotionStd.tyBtnMovRel.bRtLk				:= FALSE;
			tyP0934AW.tyAW.tyBtnGo.bRtLk						:= FALSE;
		END_IF

	ELSIF (tyP0934AW.tyMotionStd.tyBtnJogOpen.bRtCompl = TRUE) OR (tyP0934AW.tyMotionStd.tyBtnJogClose.bRtCompl = TRUE) OR (bJogStopAW = TRUE) THEN
		bJogSlow					:= FALSE;
		bJogFast					:= FALSE;
		fbJogSlowToFastDlyTm.IN		:= FALSE;

		eAWOpenAct		:= AWActJogStop;

		IF p_eAWOpenStat = AWActJogStop AND p_eAWOpenStatus = Done THEN
			eAWOpenAct	:= AWActIdle;

			bJogStopAW	:= FALSE;

			tyP0934AW.tyMotionStd.tyBtnStop.bRtCompl		:= FALSE;
			tyP0934AW.tyMotionStd.tyBtnJogOpen.bRtCompl		:= FALSE;
			tyP0934AW.tyMotionStd.tyBtnJogClose.bRtCompl	:= FALSE;
			tyP0934AW.tyMotionStd.tyBtnOrigin.bRtCompl		:= FALSE;
			tyP0934AW.tyMotionStd.tyBtnMovAbs.bRtCompl		:= FALSE;
			tyP0934AW.tyMotionStd.tyBtnMovRel.bRtCompl		:= FALSE;
			tyP0934AW.tyAW.tyBtnGo.bRtCompl					:= FALSE;

			tyP0934AW.tyMotionStd.tyBtnStop.bValue			:= TRUE;
			tyP0934AW.tyMotionStd.tyBtnJogOpen.bValue		:= FALSE;
			tyP0934AW.tyMotionStd.tyBtnJogClose.bValue		:= FALSE;
			tyP0934AW.tyMotionStd.tyBtnOrigin.bValue		:= FALSE;
			tyP0934AW.tyMotionStd.tyBtnMovAbs.bValue		:= FALSE;
			tyP0934AW.tyMotionStd.tyBtnMovRel.bValue		:= FALSE;
			tyP0934AW.tyAW.tyBtnGo.bValue					:= FALSE;

			tyP0934AW.tyMotionStd.tyBtnStop.bRtLk			:= TRUE;
			tyP0934AW.tyMotionStd.tyBtnJogOpen.bRtLk		:= FALSE;
			tyP0934AW.tyMotionStd.tyBtnJogClose.bRtLk		:= FALSE;
			tyP0934AW.tyMotionStd.tyBtnOrigin.bRtLk			:= FALSE;
			tyP0934AW.tyMotionStd.tyBtnMovAbs.bRtLk			:= FALSE;
			tyP0934AW.tyMotionStd.tyBtnMovRel.bRtLk			:= FALSE;
			tyP0934AW.tyAW.tyBtnGo.bRtLk					:= FALSE;
		END_IF

	ELSIF tyP0934AW.tyMotionStd.tyBtnPwr.bRtCompl = TRUE THEN
		tyP0934AW.tyMotionStd.tyBtnPwr.bRtLk					:= TRUE;

		IF tyP0934AW.tyMotionStd.tyBtnPwr.bValue = TRUE THEN
			eAWOpenAct		:= AWActPwrOn;

			IF p_eAWOpenStat = AWActPwrOn AND p_eAWOpenStatus = Done THEN
				eAWOpenAct	:= AWActIdle;

				tyP0934AW.tyMotionStd.tyBtnPwr.bRtCompl			:= FALSE;
				tyP0934AW.tyMotionStd.tyBtnPwr.bRtLk			:= FALSE;
			END_IF
		ELSE
			eAWOpenAct		:= AWActPwrOff;

			IF p_eAWOpenStat = AWActPwrOff AND p_eAWOpenStatus = Done THEN
				eAWOpenAct	:= AWActIdle;

				tyP0934AW.tyMotionStd.tyBtnPwr.bRtCompl			:= FALSE;
				tyP0934AW.tyMotionStd.tyBtnPwr.bRtLk			:= FALSE;
			END_IF
		END_IF

	ELSIF tyP0934AW.tyMotionStd.tyBtnOrigin.bRtCompl = TRUE THEN
		tyP0934AW.tyMotionStd.tyBtnOrigin.bValue				:= TRUE;
		tyP0934AW.tyMotionStd.tyBtnStop.bValue					:= FALSE;

		tyP0934AW.tyMotionStd.tyBtnOrigin.bRtLk					:= TRUE;
		tyP0934AW.tyMotionStd.tyBtnStop.bRtLk					:= FALSE;

		eAWOpenAct		:= AWActHoming;

		IF p_eAWOpenStat = AWActHoming AND p_eAWOpenStatus = Done THEN
			eAWOpenAct	:= AWActIdle;

			tyP0934AW.tyMotionStd.tyBtnOrigin.bRtCompl			:= FALSE;
			tyP0934AW.tyMotionStd.tyBtnOrigin.bValue			:= FALSE;
			tyP0934AW.tyMotionStd.tyBtnStop.bValue				:= TRUE;

			tyP0934AW.tyMotionStd.tyBtnOrigin.bRtLk				:= FALSE;
			tyP0934AW.tyMotionStd.tyBtnStop.bRtLk				:= TRUE;
		END_IF

	ELSIF tyP0934AW.tyMotionStd.tyBtnRst.bRtCompl = TRUE THEN
		tyP0934AW.tyMotionStd.tyBtnRst.bValue					:= TRUE;
		tyP0934AW.tyMotionStd.tyBtnRst.bRtLk					:= TRUE;

		eAWOpenAct		:= AWActRstAxisErr;

		IF p_eAWOpenStat = AWActRstAxisErr AND p_eAWOpenStatus = Done THEN
			eAWOpenAct	:= AWActIdle;

			tyP0934AW.tyMotionStd.tyBtnRst.bRtCompl				:= FALSE;
			tyP0934AW.tyMotionStd.tyBtnRst.bValue				:= FALSE;
			tyP0934AW.tyMotionStd.tyBtnRst.bRtLk				:= FALSE;

			fbLmtRstTm.IN			:= FALSE;
		END_IF

	ELSIF tyP0934AW.tyAW.tyBtnGo.bRtCompl = TRUE THEN
		tyP0934AW.tyAW.tyBtnGo.bValue							:= TRUE;
		tyP0934AW.tyMotionStd.tyBtnStop.bValue					:= FALSE;

		tyP0934AW.tyAW.tyBtnGo.bRtLk							:= TRUE;
		tyP0934AW.tyMotionStd.tyBtnStop.bRtLk					:= FALSE;

		diMnlAWGoWidth		:= tyP0934AW.tyAW.tyNumNewWidth.diValue;
		diMnlAWNomSpd		:= tyP0934AW.tyMotionStd.tyNumNomSpd.diValue;

		eAWOpenAct		:= AWActGoWidth;

		IF p_eAWOpenStat = AWActGoWidth AND p_eAWOpenStatus = Done THEN
			eAWOpenAct	:= AWActIdle;

			tyP0934AW.tyAW.tyBtnGo.bRtCompl						:= FALSE;
			tyP0934AW.tyAW.tyBtnGo.bValue						:= FALSE;
			tyP0934AW.tyMotionStd.tyBtnStop.bValue				:= TRUE;

			tyP0934AW.tyAW.tyBtnGo.bRtLk						:= FALSE;
			tyP0934AW.tyMotionStd.tyBtnStop.bRtLk				:= TRUE;
		END_IF

	ELSIF tyP0934AW.tyMotionStd.tyBtnMovAbs.bRtCompl = TRUE THEN
		tyP0934AW.tyMotionStd.tyBtnMovAbs.bValue				:= TRUE;
		tyP0934AW.tyMotionStd.tyBtnStop.bValue					:= FALSE;

		tyP0934AW.tyMotionStd.tyBtnMovAbs.bRtLk					:= TRUE;
		tyP0934AW.tyMotionStd.tyBtnStop.bRtLk					:= FALSE;

		diMnlAWTargetPos	:= tyP0934AW.tyMotionStd.tyNumTargetPos.diValue;
		diMnlAWNomSpd		:= tyP0934AW.tyMotionStd.tyNumNomSpd.diValue;

		eAWOpenAct		:= AWActMovAbs;

		IF p_eAWOpenStat = AWActMovAbs AND p_eAWOpenStatus = Done THEN
			eAWOpenAct	:= AWActIdle;

			tyP0934AW.tyMotionStd.tyBtnMovAbs.bRtCompl			:= FALSE;
			tyP0934AW.tyMotionStd.tyBtnMovAbs.bValue			:= FALSE;
			tyP0934AW.tyMotionStd.tyBtnStop.bValue				:= TRUE;

			tyP0934AW.tyMotionStd.tyBtnMovAbs.bRtLk				:= FALSE;
			tyP0934AW.tyMotionStd.tyBtnStop.bRtLk				:= TRUE;
		END_IF

	ELSIF tyP0934AW.tyMotionStd.tyBtnMovRel.bRtCompl = TRUE THEN
		tyP0934AW.tyMotionStd.tyBtnMovRel.bValue				:= TRUE;
		tyP0934AW.tyMotionStd.tyBtnStop.bValue					:= FALSE;

		tyP0934AW.tyMotionStd.tyBtnMovRel.bRtLk					:= TRUE;
		tyP0934AW.tyMotionStd.tyBtnStop.bRtLk					:= FALSE;

		diMnlAWStepSize		:= tyP0934AW.tyMotionStd.tyNumStepSize.diValue;
		diMnlAWNomSpd		:= tyP0934AW.tyMotionStd.tyNumNomSpd.diValue;

		eAWOpenAct		:= AWActMovRel;

		IF p_eAWOpenStat = AWActMovRel AND p_eAWOpenStatus = Done THEN
			eAWOpenAct	:= AWActIdle;

			tyP0934AW.tyMotionStd.tyBtnMovRel.bRtCompl			:= FALSE;
			tyP0934AW.tyMotionStd.tyBtnMovRel.bValue			:= FALSE;
			tyP0934AW.tyMotionStd.tyBtnStop.bValue				:= TRUE;

			tyP0934AW.tyMotionStd.tyBtnMovRel.bRtLk				:= FALSE;
			tyP0934AW.tyMotionStd.tyBtnStop.bRtLk				:= TRUE;
		END_IF

	ELSIF (tyP0934AW.tyMotionStd.tyBtnJogOpen.bValue = TRUE) AND (fbJogSlowToFastDlyTm.Q = FALSE) AND (bJogSlow = FALSE) THEN
		tyP0934AW.tyMotionStd.tyBtnStop.bValue					:= FALSE;
		tyP0934AW.tyMotionStd.tyBtnStop.bRtLk					:= FALSE;

		fbJogSlowToFastDlyTm.IN		:= TRUE;

		diMnlAWJogSpd	:= tyP0934AW.tyMotionStd.tyNumSlwSpd.diValue;

		eAWOpenAct		:= AWActJogOpen;

		IF p_eAWOpenStat = AWActJogOpen AND p_eAWOpenStatus = Done THEN
			eAWOpenAct				:= AWActIdle;
			bJogSlow				:= TRUE;
		ELSIF p_eAWOpenStatus = Error THEN
			fbJogSlowToFastDlyTm.IN	:= FALSE;
			bJogSlow				:= TRUE;
		END_IF

	ELSIF (tyP0934AW.tyMotionStd.tyBtnJogOpen.bValue = TRUE) AND (fbJogSlowToFastDlyTm.Q = TRUE) AND (bJogFast = FALSE) THEN
		tyP0934AW.tyMotionStd.tyBtnStop.bValue					:= FALSE;
		tyP0934AW.tyMotionStd.tyBtnStop.bRtLk					:= FALSE;

		fbJogSlowToFastDlyTm.IN		:= TRUE;

		diMnlAWJogSpd	:= tyP0934AW.tyMotionStd.tyNumNomSpd.diValue;

		eAWOpenAct		:= AWActJogOpen;

		IF p_eAWOpenStat = AWActJogOpen AND p_eAWOpenStatus = Done THEN
			eAWOpenAct				:= AWActIdle;
			bJogFast				:= TRUE;
		ELSIF p_eAWOpenStatus = Error THEN
			fbJogSlowToFastDlyTm.IN	:= FALSE;
			bJogFast				:= TRUE;
		END_IF

	ELSIF (tyP0934AW.tyMotionStd.tyBtnJogClose.bValue = TRUE) AND (fbJogSlowToFastDlyTm.Q = FALSE) AND (bJogSlow = FALSE) THEN
		tyP0934AW.tyMotionStd.tyBtnStop.bValue					:= FALSE;
		tyP0934AW.tyMotionStd.tyBtnStop.bRtLk					:= FALSE;

		fbJogSlowToFastDlyTm.IN		:= TRUE;

		diMnlAWJogSpd	:= tyP0934AW.tyMotionStd.tyNumSlwSpd.diValue;

		eAWOpenAct		:= AWActJogClose;

		IF p_eAWOpenStat = AWActJogClose AND p_eAWOpenStatus = Done THEN
			eAWOpenAct				:= AWActIdle;
			bJogSlow				:= TRUE;
		ELSIF p_eAWOpenStatus = Error THEN
			fbJogSlowToFastDlyTm.IN	:= FALSE;
			bJogSlow				:= TRUE;
		END_IF

	ELSIF (tyP0934AW.tyMotionStd.tyBtnJogClose.bValue = TRUE) AND (fbJogSlowToFastDlyTm.Q = TRUE) AND (bJogFast = FALSE) THEN
		tyP0934AW.tyMotionStd.tyBtnStop.bValue					:= FALSE;
		tyP0934AW.tyMotionStd.tyBtnStop.bRtLk					:= FALSE;

		fbJogSlowToFastDlyTm.IN		:= TRUE;

		diMnlAWJogSpd	:= tyP0934AW.tyMotionStd.tyNumNomSpd.diValue;

		eAWOpenAct		:= AWActJogClose;

		IF p_eAWOpenStat = AWActJogClose AND p_eAWOpenStatus = Done THEN
			eAWOpenAct				:= AWActIdle;
			bJogFast				:= TRUE;
		ELSIF p_eAWOpenStatus = Error THEN
			fbJogSlowToFastDlyTm.IN	:= FALSE;
			bJogFast				:= TRUE;
		END_IF

	END_IF

END_ACTION
```

#### Act_OptP0934FBStat.st
```iecst
ACTION Act_OptP0934FBStat:

	IF p_bAWOpenAxisErr = TRUE THEN
		tyP0934AW.tyMotionStd.tyStringStat.sValue	:= p_sAWOpenAxisErrTxt;
	ELSE
		IF NOT (p_bAWOpenJogging AND p_eAWOpenStat = AWActIdle) THEN

			tyP0934AW.tyMotionStd.tyStringStat.sValue	:= p_sAWOpenStatTxt;
		END_IF

	END_IF

END_ACTION
```

#### Act_OptP0934Mask.st
```iecst
ACTION Act_OptP0934Mask:

	//Interlock Power
	IF p_bAWOpenAxisErr = TRUE AND p_bAWOpenPwrOn = FALSE THEN
		tyP0934AW.tyMotionStd.tyBtnPwr.bValue		:= FALSE;

		fUIInRtStatOff(ADR(tyP0934AW.tyMotionStd.tyBtnPwr.uiMaskRtStat));
	ELSE
		fUIInRtStatHide(ADR(tyP0934AW.tyMotionStd.tyBtnPwr.uiMaskRtStat));
	END_IF

	//Interlock Others Move
	IF p_bAWOpenAxisErr = TRUE OR p_bAWOpenPwrOn = FALSE THEN
		fUIInRtStatOff(ADR(tyP0934AW.tyMotionStd.tyBtnOrigin.uiMaskRtStat));
		fUIInRtStatOff(ADR(tyP0934AW.tyMotionStd.tyBtnMovRel.uiMaskRtStat));
		fUIInRtStatOff(ADR(tyP0934AW.tyMotionStd.tyBtnJogOpen.uiMaskRtStat));
		fUIInRtStatOff(ADR(tyP0934AW.tyMotionStd.tyBtnJogClose.uiMaskRtStat));
	ELSE
		fUIInRtStatHide(ADR(tyP0934AW.tyMotionStd.tyBtnOrigin.uiMaskRtStat));
		fUIInRtStatHide(ADR(tyP0934AW.tyMotionStd.tyBtnMovRel.uiMaskRtStat));
		fUIInRtStatHide(ADR(tyP0934AW.tyMotionStd.tyBtnJogOpen.uiMaskRtStat));
		fUIInRtStatHide(ADR(tyP0934AW.tyMotionStd.tyBtnJogClose.uiMaskRtStat));
	END_IF

	//Interlock Move Absolute
	IF p_bAWOpenAxisErr = TRUE OR p_bAWOpenPwrOn = FALSE OR p_bAWOpenIsHomed = FALSE THEN
		fUIInRtStatOff(ADR(tyP0934AW.tyAW.tyBtnGo.uiMaskRtStat));
		fUIInRtStatOff(ADR(tyP0934AW.tyMotionStd.tyBtnMovAbs.uiMaskRtStat));
	ELSE
		fUIInRtStatHide(ADR(tyP0934AW.tyAW.tyBtnGo.uiMaskRtStat));
		fUIInRtStatHide(ADR(tyP0934AW.tyMotionStd.tyBtnMovAbs.uiMaskRtStat));
	END_IF

	//Interlock Limit Sensor
	IF tyP0934AW.tyMotionStd.tyBtnOpenLmtSen.bValue = TRUE THEN
		fUIInRtStatOff(ADR(tyP0934AW.tyMotionStd.tyBtnJogOpen.uiMaskRtStat));
	END_IF

	IF tyP0934AW.tyMotionStd.tyBtnCloseLmtSen.bValue = TRUE THEN
		fUIInRtStatOff(ADR(tyP0934AW.tyMotionStd.tyBtnJogClose.uiMaskRtStat));
	END_IF

	//Interlock When Moving
	IF tyP0934AW.tyMotionStd.tyBtnOrigin.bRtCompl = TRUE THEN
		fUIInRtStatOff(ADR(tyP0934AW.tyMotionStd.tyBtnMovAbs.uiMaskRtStat));
		fUIInRtStatOff(ADR(tyP0934AW.tyMotionStd.tyBtnMovRel.uiMaskRtStat));
		fUIInRtStatOff(ADR(tyP0934AW.tyMotionStd.tyBtnJogOpen.uiMaskRtStat));
		fUIInRtStatOff(ADR(tyP0934AW.tyMotionStd.tyBtnJogClose.uiMaskRtStat));
		fUIInRtStatOff(ADR(tyP0934AW.tyAW.tyBtnGo.uiMaskRtStat));

	ELSIF tyP0934AW.tyMotionStd.tyBtnMovAbs.bRtCompl = TRUE THEN
		fUIInRtStatOff(ADR(tyP0934AW.tyMotionStd.tyBtnOrigin.uiMaskRtStat));
		fUIInRtStatOff(ADR(tyP0934AW.tyMotionStd.tyBtnMovRel.uiMaskRtStat));
		fUIInRtStatOff(ADR(tyP0934AW.tyMotionStd.tyBtnJogOpen.uiMaskRtStat));
		fUIInRtStatOff(ADR(tyP0934AW.tyMotionStd.tyBtnJogClose.uiMaskRtStat));
		fUIInRtStatOff(ADR(tyP0934AW.tyAW.tyBtnGo.uiMaskRtStat));

	ELSIF tyP0934AW.tyMotionStd.tyBtnMovRel.bRtCompl = TRUE THEN
		fUIInRtStatOff(ADR(tyP0934AW.tyMotionStd.tyBtnOrigin.uiMaskRtStat));
		fUIInRtStatOff(ADR(tyP0934AW.tyMotionStd.tyBtnMovAbs.uiMaskRtStat));
		fUIInRtStatOff(ADR(tyP0934AW.tyMotionStd.tyBtnJogOpen.uiMaskRtStat));
		fUIInRtStatOff(ADR(tyP0934AW.tyMotionStd.tyBtnJogClose.uiMaskRtStat));
		fUIInRtStatOff(ADR(tyP0934AW.tyAW.tyBtnGo.uiMaskRtStat));

	ELSIF (tyP0934AW.tyMotionStd.tyBtnJogOpen.bRtCompl = TRUE) OR (tyP0934AW.tyMotionStd.tyBtnJogOpen.bValue = TRUE) THEN
		fUIInRtStatOff(ADR(tyP0934AW.tyMotionStd.tyBtnOrigin.uiMaskRtStat));
		fUIInRtStatOff(ADR(tyP0934AW.tyMotionStd.tyBtnMovAbs.uiMaskRtStat));
		fUIInRtStatOff(ADR(tyP0934AW.tyMotionStd.tyBtnMovRel.uiMaskRtStat));
		fUIInRtStatOff(ADR(tyP0934AW.tyMotionStd.tyBtnJogClose.uiMaskRtStat));
		fUIInRtStatOff(ADR(tyP0934AW.tyAW.tyBtnGo.uiMaskRtStat));

	ELSIF (tyP0934AW.tyMotionStd.tyBtnJogClose.bRtCompl = TRUE) OR (tyP0934AW.tyMotionStd.tyBtnJogClose.bValue = TRUE) THEN
		fUIInRtStatOff(ADR(tyP0934AW.tyMotionStd.tyBtnOrigin.uiMaskRtStat));
		fUIInRtStatOff(ADR(tyP0934AW.tyMotionStd.tyBtnMovAbs.uiMaskRtStat));
		fUIInRtStatOff(ADR(tyP0934AW.tyMotionStd.tyBtnMovRel.uiMaskRtStat));
		fUIInRtStatOff(ADR(tyP0934AW.tyMotionStd.tyBtnJogOpen.uiMaskRtStat));
		fUIInRtStatOff(ADR(tyP0934AW.tyAW.tyBtnGo.uiMaskRtStat));

	ELSIF tyP0934AW.tyAW.tyBtnGo.bRtCompl = TRUE THEN
		fUIInRtStatOff(ADR(tyP0934AW.tyMotionStd.tyBtnOrigin.uiMaskRtStat));
		fUIInRtStatOff(ADR(tyP0934AW.tyMotionStd.tyBtnMovAbs.uiMaskRtStat));
		fUIInRtStatOff(ADR(tyP0934AW.tyMotionStd.tyBtnMovRel.uiMaskRtStat));
		fUIInRtStatOff(ADR(tyP0934AW.tyMotionStd.tyBtnJogOpen.uiMaskRtStat));
		fUIInRtStatOff(ADR(tyP0934AW.tyMotionStd.tyBtnJogClose.uiMaskRtStat));

	END_IF

	//Axis Error
	IF tyP0934AW.tyMotionStd.tyBtnPwr.bRtCompl = TRUE  THEN
		fUIInRtStatOff(ADR(tyP0934AW.tyMotionStd.tyBtnRst.uiMaskRtStat));
	ELSE
		fUIInRtStatHide(ADR(tyP0934AW.tyMotionStd.tyBtnRst.uiMaskRtStat));
	END_IF

END_ACTION
```

#### Act_OptP0934UpdtDat.st
```iecst
ACTION Act_OptP0934UpdtDat:

	tyP0934AW.tyMotionStd.tyNumCurrPos.diValue			:= p_diAWOpenActualPos;
	tyP0934AW.tyMotionStd.tyNumErrCode.diValue			:= UDINT_TO_DINT(p_udiAWOpenAxisErrID);
	tyP0934AW.tyMotionStd.tyBitmapPwr.usiValueIdx		:= BOOL_TO_USINT(p_bAWOpenPwrOn);
	tyP0934AW.tyMotionStd.tyBitmapRst.usiValueIdx		:= BOOL_TO_USINT(NOT p_bAWOpenAxisErr);
	tyP0934AW.tyMotionStd.tyBitmapOrigin.usiValueIdx	:= BOOL_TO_USINT(p_bAWOpenIsHomed);

	tyP0934AW.tyMotionStd.tyBtnOpenLmtSen.bValue		:= p_bAWOpenOpenSen;
	tyP0934AW.tyMotionStd.tyBtnCloseLmtSen.bValue		:= p_bAWOpenCloseSen;

	//Bitmap Machine
	IF p_tyNtParamCurr.tyDOSettings.diTLGreen<>0 OR p_tyNtParamCurr.tyDOSettings.diTLAmber<>0 OR p_tyNtParamCurr.tyDOSettings.diTLRed<>0 THEN
		IF p_tyNtParamCurr.eTLBuzMode=TLBuzModBHTC THEN
			IF p_bAWOpenIsHomed = TRUE THEN
				IF p_diAWOpenActualPos <= (p_tyNtParamCurr.tyProdRcpWidthLmt.diMax / 2) THEN
					tyP0934AW.tyMotionStd.tyBitmapMc.usiValueIdx	:= 200;
				ELSE
					tyP0934AW.tyMotionStd.tyBitmapMc.usiValueIdx	:= 201;
				END_IF
			ELSE
				tyP0934AW.tyMotionStd.tyBitmapMc.usiValueIdx	:= 200;
			END_IF
		ELSE
			IF p_bAWOpenIsHomed = TRUE THEN
				IF p_diAWOpenActualPos <= (p_tyNtParamCurr.tyProdRcpWidthLmt.diMax / 2) THEN
					tyP0934AW.tyMotionStd.tyBitmapMc.usiValueIdx	:= 100;
				ELSE
					tyP0934AW.tyMotionStd.tyBitmapMc.usiValueIdx	:= 101;
				END_IF
			ELSE
				tyP0934AW.tyMotionStd.tyBitmapMc.usiValueIdx	:= 100;
			END_IF
		END_IF
	ELSE
		IF p_bAWOpenIsHomed = TRUE THEN
			IF p_diAWOpenActualPos <= (p_tyNtParamCurr.tyProdRcpWidthLmt.diMax / 2) THEN
				tyP0934AW.tyMotionStd.tyBitmapMc.usiValueIdx	:= 0;
			ELSE
				tyP0934AW.tyMotionStd.tyBitmapMc.usiValueIdx	:= 1;
			END_IF
		ELSE
			tyP0934AW.tyMotionStd.tyBitmapMc.usiValueIdx	:= 0;
		END_IF
	END_IF

END_ACTION
```

#### Act_OptP0934Keypad.st
```iecst
ACTION Act_OptP0934Keypad:

	IF fUIOutRtStatTPIsOpen(ADR(tyP0934AW.tyAW.tyNumNewWidth.uiRtStat)) = TRUE THEN
		tyProperty.tyKeypad.tyTxtTitle.sTxt		:= tyP0934AW.tyAW.tyNumNewWidth.sKeypadTitle;

	ELSIF fUIOutRtStatTPIsOpen(ADR(tyP0934AW.tyMotionStd.tyNumTargetPos.uiRtStat)) = TRUE THEN
		tyProperty.tyKeypad.tyTxtTitle.sTxt		:= tyP0934AW.tyMotionStd.tyNumTargetPos.sKeypadTitle;

	ELSIF fUIOutRtStatTPIsOpen(ADR(tyP0934AW.tyMotionStd.tyNumStepSize.uiRtStat)) = TRUE THEN
		tyProperty.tyKeypad.tyTxtTitle.sTxt		:= tyP0934AW.tyMotionStd.tyNumStepSize.sKeypadTitle;

	ELSIF fUIOutRtStatTPIsOpen(ADR(tyP0934AW.tyMotionStd.tyNumNomSpd.uiRtStat)) = TRUE THEN
		tyProperty.tyKeypad.tyTxtTitle.sTxt		:= tyP0934AW.tyMotionStd.tyNumNomSpd.sKeypadTitle;

	ELSIF fUIOutRtStatTPIsOpen(ADR(tyP0934AW.tyMotionStd.tyNumSlwSpd.uiRtStat)) = TRUE THEN
		tyProperty.tyKeypad.tyTxtTitle.sTxt		:= tyP0934AW.tyMotionStd.tyNumSlwSpd.sKeypadTitle;

	END_IF

END_ACTION
```

#### Act_OptP0934RstMnl.st
```iecst
ACTION Act_OptP0934RstMnl:

	IF EDGEPOS((bManualMod = FALSE) OR (p_eAWOpenStatus = Error)) THEN

		eAWOpenAct	:= AWActIdle;

		bJogSlow					:= FALSE;
		bJogFast					:= FALSE;
		fbJogSlowToFastDlyTm.IN		:= FALSE;

		tyP0934AW.tyAW.tyBtnGo.bRtCompl					:= FALSE;
		tyP0934AW.tyAW.tyBtnGo.bValue					:= FALSE;
		tyP0934AW.tyAW.tyBtnGo.bRtLk					:= FALSE;
		tyP0934AW.tyAW.tyBtnGo.uiMaskRtStat.0			:= FALSE;

		tyP0934AW.tyMotionStd.tyBtnPwr.bRtCompl				:= FALSE;
		tyP0934AW.tyMotionStd.tyBtnStop.bRtCompl			:= FALSE;
		tyP0934AW.tyMotionStd.tyBtnOrigin.bRtCompl			:= FALSE;
		tyP0934AW.tyMotionStd.tyBtnRst.bRtCompl				:= FALSE;
		tyP0934AW.tyMotionStd.tyBtnMovAbs.bRtCompl			:= FALSE;
		tyP0934AW.tyMotionStd.tyBtnMovRel.bRtCompl			:= FALSE;
		tyP0934AW.tyMotionStd.tyBtnJogOpen.bRtCompl			:= FALSE;
		tyP0934AW.tyMotionStd.tyBtnJogClose.bRtCompl		:= FALSE;

		tyP0934AW.tyMotionStd.tyBtnPwr.bValue				:= FALSE;
		tyP0934AW.tyMotionStd.tyBtnStop.bValue				:= TRUE;
		tyP0934AW.tyMotionStd.tyBtnOrigin.bValue			:= FALSE;
		tyP0934AW.tyMotionStd.tyBtnRst.bValue				:= FALSE;
		tyP0934AW.tyMotionStd.tyBtnMovAbs.bValue			:= FALSE;
		tyP0934AW.tyMotionStd.tyBtnMovRel.bValue			:= FALSE;
		tyP0934AW.tyMotionStd.tyBtnJogOpen.bValue			:= FALSE;
		tyP0934AW.tyMotionStd.tyBtnJogClose.bValue			:= FALSE;

		tyP0934AW.tyMotionStd.tyBtnPwr.bRtLk				:= FALSE;
		tyP0934AW.tyMotionStd.tyBtnStop.bRtLk				:= TRUE;
		tyP0934AW.tyMotionStd.tyBtnOrigin.bRtLk				:= FALSE;
		tyP0934AW.tyMotionStd.tyBtnRst.bRtLk				:= FALSE;
		tyP0934AW.tyMotionStd.tyBtnMovAbs.bRtLk				:= FALSE;
		tyP0934AW.tyMotionStd.tyBtnMovRel.bRtLk				:= FALSE;
		tyP0934AW.tyMotionStd.tyBtnJogOpen.bRtLk			:= FALSE;
		tyP0934AW.tyMotionStd.tyBtnJogClose.bRtLk			:= FALSE;

		tyP0934AW.tyMotionStd.tyBtnPwr.uiMaskRtStat			:= TRUE;
		tyP0934AW.tyMotionStd.tyBtnOrigin.uiMaskRtStat		:= FALSE;
		tyP0934AW.tyMotionStd.tyBtnRst.uiMaskRtStat			:= TRUE;
		tyP0934AW.tyMotionStd.tyBtnMovAbs.uiMaskRtStat		:= FALSE;
		tyP0934AW.tyMotionStd.tyBtnMovRel.uiMaskRtStat		:= FALSE;
		tyP0934AW.tyMotionStd.tyBtnJogOpen.uiMaskRtStat		:= FALSE;
		tyP0934AW.tyMotionStd.tyBtnJogClose.uiMaskRtStat	:= FALSE;

	END_IF

END_ACTION
```
